legal notes
=================
| SPDX-FileCopyrightText: © 2022 ekvip automation GmbH <info@ekvip.de>
| SPDX-License-Identifier: Apache-2.0
| For details check: Apache-2.0_

.. _Apache-2.0: https://www.apache.org/licenses/LICENSE-2.0

.. _Apache-2.THIS^.SIZE_ZERO: https://www.apache.org/licenses/LICENSE-2.THIS^.SIZE_ZERO

.. </legal notes>

*)

METHOD runIsDwordAlignedTests
VAR
	foo				:XWORD;
	stackAddress	:PVOID;
END_VAR
VAR CONSTANT
	aDWord :DWORD := 16#4;
END_VAR
RETURN (NOT TcUnit.TEST_ORDERED(THIS^.getTestNameFor('isDwordAligned')));
stackAddress := ADR(foo);

THIS^.testIsDwordAligned(
	address := THIS,
);
THIS^.testIsDwordAligned(
	address := THIS^.NULL_POINTER,
);
THIS^.testIsDwordAligned(
	address := THIS^.NULL_POINTER + 1,
);
THIS^.testIsDwordAligned(
	address := stackAddress,
);
THIS^.testIsDwordAligned(
	address := stackAddress + 3,
);
THIS^.testIsDwordAligned(
	address := THIS^.oneByte,
);
THIS^.testIsDwordAligned(
	address := THIS^.oneByte + 7,
);
THIS^.testIsDwordAligned(
	address := THIS^.byteArray,
);
THIS^.testIsDwordAligned(
	address := THIS^.byteArray + 2,
);
THIS^.testIsDwordAligned(
	address := THIS^.cncAddress,
);
THIS^.testIsDwordAligned(
	address := THIS^.cncAddress + 1,
);
THIS^.testIsDwordAligned(
	address := THIS^.itsMeAgain,
);
THIS^.testIsDwordAligned(
	address := THIS^.itsMeAgain + 6,
);
THIS^.testIsDwordAligned(
	address := THIS^.me,
);
THIS^.testIsDwordAligned(
	address := THIS^.me + 3,
);
THIS^.testIsDwordAligned(
	address := THIS^.myMom,
);
THIS^.testIsDwordAligned(
	address := THIS^.invalidByte,
);
THIS^.testIsDwordAligned(
	address := THIS^.invalidByte + 4,
);
THIS^.testIsDwordAligned(
	address := THIS^.INVALID_POINTER,
);
THIS^.testIsDwordAligned(
	address := THIS^.INVALID_POINTER + 1,
);
THIS^.testIsDwordAligned(
	address := aDWord,
);
THIS^.testIsDwordAligned(
	address := aDWord + 1,
);
THIS^.testIsDwordAligned(
	address := TO_DWORD(aDWord - 1),
);

TcUnit.TEST_FINISHED();
END_METHOD

(*

short summary
==================
This test method tests ``assert.pointers.isEqualTo``
method of CNM_AssertionInterfaces library with various inputs

.. <legal notes>

legal notes
=================
| SPDX-FileCopyrightText: © 2022 ekvip automation GmbH <info@ekvip.de>
| SPDX-License-Identifier: Apache-2.0
| For details check: Apache-2.0_

.. _Apache-2.0: https://www.apache.org/licenses/LICENSE-2.0

.. </legal notes>

*)

METHOD runIsEqualToTests
VAR
	foo				:__XWORD;
	stackAddress	:PVOID;
END_VAR
RETURN (NOT TcUnit.TEST_ORDERED(THIS^.getTestNameFor('isEqualTo')));
stackAddress := ADR(foo);
THIS^.testIsEqualTo(
	address1 := THIS,
	address2 := THIS
);
THIS^.testIsEqualTo(
	address1 := THIS^.NULL_POINTER,
	address2 := THIS^.NULL_POINTER
);
THIS^.testIsEqualTo(
	address1 := stackAddress,
	address2 := stackAddress
);
THIS^.testIsEqualTo(
	address1 := THIS^.oneByte,
	address2 := THIS^.oneByte
);
THIS^.testIsEqualTo(
	address1 := THIS^.byteArray,
	address2 := THIS^.byteArray
);
THIS^.testIsEqualTo(
	address1 := THIS^.cncAddress,
	address2 := THIS^.cncAddress
);
THIS^.testIsEqualTo(
	address1 := THIS^.itsMeAgain,
	address2 := THIS^.itsMeAgain
);
THIS^.testIsEqualTo(
	address1 := THIS^.itsMeAgain^,
	address2 := THIS^.itsMeAgain^
);
THIS^.testIsEqualTo(
	address1 := THIS^.me,
	address2 := THIS
);

THIS^.testIsEqualTo(
	address1 := THIS^.itsMeAgain,
	address2 := THIS
);
THIS^.testIsEqualTo(
	address1 := THIS,
	address2 := THIS^.NULL_POINTER
);
THIS^.testIsEqualTo(
	address1 := THIS^.NULL_POINTER,
	address2 := stackAddress
);
THIS^.testIsEqualTo(
	address1 := stackAddress,
	address2 := THIS^.oneByte
);
THIS^.testIsEqualTo(
	address1 := THIS^.oneByte,
	address2 := THIS^.byteArray
);
THIS^.testIsEqualTo(
	address1 := THIS^.byteArray,
	address2 := THIS^.cncAddress
);
THIS^.testIsEqualTo(
	address1 := THIS^.itsMeAgain,
	address2 := THIS^.itsMeAgain
);
THIS^.testIsEqualTo(
	address1 := THIS^.cncAddress,
	address2 := THIS^.itsMeAgain^
);
THIS^.testIsEqualTo(
	address1 := THIS^.itsMeAgain^,
	address2 := THIS^.itsMeAgain
);
THIS^.testIsEqualTo(
	address1 := THIS^.itsMeAgain,
	address2 := THIS
);

TcUnit.TEST_FINISHED();
END_METHOD

(*

short summary
==================
This test method tests ``assert.pointers.isLwordAligned``
method of CNM_AssertionInterfaces library with various inputs

.. <legal notes>

legal notes
=================
| SPDX-FileCopyrightText: © 2022 ekvip automation GmbH <info@ekvip.de>
| SPDX-License-Identifier: Apache-2.0
| For details check: Apache-2.0_

.. _Apache-2.0: https://www.apache.org/licenses/LICENSE-2.0

.. _Apache-2.THIS^.SIZE_ZERO: https://www.apache.org/licenses/LICENSE-2.THIS^.SIZE_ZERO

.. </legal notes>

*)

METHOD runIsLwordAlignedTests
VAR
	foo				:XWORD;
	stackAddress	:PVOID;
	anLword :DWORD := 16#8;
END_VAR
RETURN (NOT TcUnit.TEST_ORDERED(THIS^.getTestNameFor('isLwordAligned')));
stackAddress := ADR(foo);

THIS^.testIsLwordAligned(
	address := THIS,
);
THIS^.testIsLwordAligned(
	address := THIS^.NULL_POINTER,
);
THIS^.testIsLwordAligned(
	address := THIS^.NULL_POINTER + 1,
);
THIS^.testIsLwordAligned(
	address := stackAddress,
);
THIS^.testIsLwordAligned(
	address := stackAddress + 3,
);
THIS^.testIsLwordAligned(
	address := THIS^.oneByte,
);
THIS^.testIsLwordAligned(
	address := THIS^.oneByte + 7,
);
THIS^.testIsLwordAligned(
	address := THIS^.byteArray,
);
THIS^.testIsLwordAligned(
	address := THIS^.byteArray + 2,
);
THIS^.testIsLwordAligned(
	address := THIS^.cncAddress,
);
THIS^.testIsLwordAligned(
	address := THIS^.cncAddress + 1,
);
THIS^.testIsLwordAligned(
	address := THIS^.itsMeAgain,
);
THIS^.testIsLwordAligned(
	address := THIS^.itsMeAgain + 6,
);
THIS^.testIsLwordAligned(
	address := THIS^.me,
);
THIS^.testIsLwordAligned(
	address := THIS^.me + 3,
);
THIS^.testIsLwordAligned(
	address := THIS^.myMom,
);
THIS^.testIsLwordAligned(
	address := THIS^.invalidByte,
);
THIS^.testIsLwordAligned(
	address := THIS^.invalidByte + 4,
);
THIS^.testIsLwordAligned(
	address := THIS^.INVALID_POINTER,
);
THIS^.testIsLwordAligned(
	address := THIS^.INVALID_POINTER + 1,
);
THIS^.testIsLwordAligned(
	address := anLword,
);
THIS^.testIsLwordAligned(
	address := anLword + 1,
);
THIS^.testIsLwordAligned(
	address := anLword - 1,
);

TcUnit.TEST_FINISHED();
END_METHOD

(*

short summary
==================
This test method tests ``assert.pointers.isNotEqualTo``
method of CNM_AssertionInterfaces library with various inputs

.. <legal notes>

legal notes
=================
| SPDX-FileCopyrightText: © 2022 ekvip automation GmbH <info@ekvip.de>
| SPDX-License-Identifier: Apache-2.0
| For details check: Apache-2.0_

.. _Apache-2.0: https://www.apache.org/licenses/LICENSE-2.0

.. </legal notes>

*)

METHOD runIsNotEqualToTests
VAR
	foo				:__XWORD;
	stackAddress	:PVOID;
END_VAR
RETURN (NOT TcUnit.TEST_ORDERED(THIS^.getTestNameFor('isNotEqualTo')));
stackAddress := ADR(foo);
THIS^.testNotIsEqualTo(
	address1 := THIS,
	address2 := THIS
);
THIS^.testNotIsEqualTo(
	address1 := THIS^.NULL_POINTER,
	address2 := THIS^.NULL_POINTER
);
THIS^.testNotIsEqualTo(
	address1 := stackAddress,
	address2 := stackAddress
);
THIS^.testNotIsEqualTo(
	address1 := THIS^.oneByte,
	address2 := THIS^.oneByte
);
THIS^.testNotIsEqualTo(
	address1 := THIS^.byteArray,
	address2 := THIS^.byteArray
);
THIS^.testNotIsEqualTo(
	address1 := THIS^.cncAddress,
	address2 := THIS^.cncAddress
);
THIS^.testNotIsEqualTo(
	address1 := THIS^.itsMeAgain,
	address2 := THIS^.itsMeAgain
);
THIS^.testNotIsEqualTo(
	address1 := THIS^.itsMeAgain^,
	address2 := THIS^.itsMeAgain^
);
THIS^.testNotIsEqualTo(
	address1 := THIS^.me,
	address2 := THIS
);

THIS^.testNotIsEqualTo(
	address1 := THIS^.itsMeAgain,
	address2 := THIS
);
THIS^.testNotIsEqualTo(
	address1 := THIS,
	address2 := THIS^.NULL_POINTER
);
THIS^.testNotIsEqualTo(
	address1 := THIS^.NULL_POINTER,
	address2 := stackAddress
);
THIS^.testNotIsEqualTo(
	address1 := stackAddress,
	address2 := THIS^.oneByte
);
THIS^.testNotIsEqualTo(
	address1 := THIS^.oneByte,
	address2 := THIS^.byteArray
);
THIS^.testNotIsEqualTo(
	address1 := THIS^.byteArray,
	address2 := THIS^.cncAddress
);
THIS^.testNotIsEqualTo(
	address1 := THIS^.itsMeAgain,
	address2 := THIS^.itsMeAgain
);
THIS^.testNotIsEqualTo(
	address1 := THIS^.cncAddress,
	address2 := THIS^.itsMeAgain^
);
THIS^.testNotIsEqualTo(
	address1 := THIS^.itsMeAgain^,
	address2 := THIS^.itsMeAgain
);
THIS^.testNotIsEqualTo(
	address1 := THIS^.itsMeAgain,
	address2 := THIS
);

TcUnit.TEST_FINISHED();
END_METHOD

(*

short summary
==================
This test method tests ``assert.pointers.isNotNull``
method of CNM_AssertionInterfaces library with various inputs

.. <legal notes>

legal notes
=================
| SPDX-FileCopyrightText: © 2022 ekvip automation GmbH <info@ekvip.de>
| SPDX-License-Identifier: Apache-2.0
| For details check: Apache-2.0_

.. _Apache-2.0: https://www.apache.org/licenses/LICENSE-2.0

.. </legal notes>

*)

METHOD runIsNotNullTests
VAR
	foo				:__XWORD;
	stackAddress	:PVOID;
END_VAR
RETURN (NOT TcUnit.TEST_ORDERED(THIS^.getTestNameFor('isNotNull')));

stackAddress := ADR(foo);

THIS^.testIsNotNull(
	address := THIS,
	symbol := 'THIS'
);
THIS^.testIsNotNull(
	address := THIS^.NULL_POINTER,
	symbol := 'THIS^.NULL_POINTER'
);
THIS^.testIsNotNull(
	address := stackAddress,
	symbol := 'stackAddress'
);
THIS^.testIsNotNull(
	address := THIS^.oneByte,
	symbol := 'THIS^.oneByte'
);
THIS^.testIsNotNull(
	address := THIS^.byteArray,
	symbol := 'THIS^.byteArray'
);
THIS^.testIsNotNull(
	address := THIS^.cncAddress,
	symbol := 'THIS^.cncAddress'
);
THIS^.testIsNotNull(
	address := THIS^.itsMeAgain,
	symbol := 'THIS^.itsMeAgain'
);
THIS^.testIsNotNull(
	address := THIS^.itsMeAgain^,
	symbol := 'THIS^.itsMeAgain^'
);
THIS^.testIsNotNull(
	address := THIS^.me,
	symbol := 'THIS^.me'
);

TcUnit.TEST_FINISHED();
END_METHOD

(*

short summary
==================
This test method tests ``assert.pointers.isNotOverlapping``
method of CNM_AssertionInterfaces library with various inputs

.. <legal notes>

legal notes
=================
| SPDX-FileCopyrightText: © 2022 ekvip automation GmbH <info@ekvip.de>
| SPDX-License-Identifier: Apache-2.0
| For details check: Apache-2.0_

.. _Apache-2.0: https://www.apache.org/licenses/LICENSE-2.0

.. _Apache-2.THIS^.SIZE_ZERO: https://www.apache.org/licenses/LICENSE-2.THIS^.SIZE_ZERO

.. </legal notes>

*)

METHOD runIsNotOverlappingTests
VAR
	foo				:XWORD;
	stackAddress	:PVOID;
END_VAR
RETURN (NOT TcUnit.TEST_ORDERED(THIS^.getTestNameFor('isNotOverlapping')));
stackAddress := ADR(foo);

THIS^.testisNotOverlapping(
	address1 := THIS,
	sizeInBytes1 := THIS^.I_AM_FAT,
	address2 := THIS,
	sizeInBytes2 := THIS^.I_AM_FAT
);
THIS^.testisNotOverlapping(
	address1 := THIS,
	sizeInBytes1 := THIS^.I_AM_FAT,
	address2 := THIS^.NULL_POINTER,
	sizeInBytes2 := THIS^.SIZE_ZERO
);
THIS^.testisNotOverlapping(
	address1 := THIS^.NULL_POINTER,
	sizeInBytes1 := THIS^.SIZE_ZERO,
	address2 := THIS^.NULL_POINTER,
	sizeInBytes2 := THIS^.SIZE_ZERO
);
THIS^.testisNotOverlapping(
	address1 := THIS^.NULL_POINTER,
	sizeInBytes1 := THIS^.SIZE_ZERO + 1,
	address2 := THIS^.NULL_POINTER + 1,
	sizeInBytes2 := THIS^.SIZE_ZERO
);
THIS^.testisNotOverlapping(
	address1 := stackAddress,
	sizeInBytes1 := THIS^.SIZE_ZERO,
	address2 := THIS^.oneByte,
	sizeInBytes2 := SIZEOF(BYTE)
);
THIS^.testisNotOverlapping(
	address1 := stackAddress,
	sizeInBytes1 := THIS^.SIZE_ZERO,
	address2 := stackAddress + 1,
	sizeInBytes2 := THIS^.SIZE_ZERO
);
THIS^.testisNotOverlapping(
	address1 := THIS^.byteArray,
	sizeInBytes1 := THIS^.ARRAY_SIZE,
	address2 := THIS^.byteArray + SIZEOF(BYTE),
	sizeInBytes2 := THIS^.SIZE_ZERO
);
THIS^.testisNotOverlapping(
	address2 := THIS^.byteArray,
	sizeInBytes2 := THIS^.ARRAY_SIZE,
	address1 := THIS^.byteArray,
	sizeInBytes1 := THIS^.ARRAY_SIZE + SIZEOF(BYTE)
);
THIS^.testisNotOverlapping(
	address1 := THIS^.cncAddress,
	sizeInBytes1 := THIS^.cncSize,
	address2 := THIS^.cncAddress,
	sizeInBytes2 := THIS^.cncSize,
);
THIS^.testisNotOverlapping(
	address1 := THIS^.cncAddress,
	sizeInBytes1 := THIS^.cncSize - 2,
	address2 := THIS^.cncAddress + 2,
	sizeInBytes2 := THIS^.cncSize + 2,
);
THIS^.testisNotOverlapping(
	address1 := THIS^.itsMeAgain,
	sizeInBytes1 := THIS^.I_AM_FAT,
	address2 := THIS,
	sizeInBytes2 := THIS^.I_AM_FAT
);
THIS^.testisNotOverlapping(
	address1 := THIS^.itsMeAgain,
	sizeInBytes1 := THIS^.I_AM_FAT,
	address2 := THIS^.me,
	sizeInBytes2 := THIS^.I_AM_FAT
);
THIS^.testisNotOverlapping(
	address1 := THIS^.itsMeAgain + 2 * SIZEOF(BYTE),
	sizeInBytes1 := THIS^.I_AM_FAT,
	address2 := THIS^.me,
	sizeInBytes2 := THIS^.I_AM_FAT
);
THIS^.testisNotOverlapping(
	address1 := THIS^.myMom,
	sizeInBytes1 := SIZEOF(AbstractAssertorTest),
	address2 := THIS^.me,
	sizeInBytes2 := THIS^.I_AM_FAT
);
THIS^.testisNotOverlapping(
	address1 := THIS^.myMom,
	sizeInBytes1 := SIZEOF(AbstractAssertorTest),
	address2 := THIS^.me,
	sizeInBytes2 := SIZEOF(AbstractAssertorTest) - THIS^.I_AM_FAT
);
THIS^.testisNotOverlapping(
	address1 := THIS^.invalidByte,
	sizeInBytes1 := SIZEOF(BYTE),
	address2 := THIS^.invalidByte,
	sizeInBytes2 := SIZEOF(BYTE)
);
THIS^.testisNotOverlapping(
	address1 := THIS^.invalidByte,
	sizeInBytes1 := SIZEOF(BYTE),
	address2 := THIS^.invalidByte + (2 * SIZEOF(BYTE)),
	sizeInBytes2 := SIZEOF(BYTE)
);
THIS^.testisNotOverlapping(
	address1 := THIS^.INVALID_POINTER,
	sizeInBytes1 := SIZEOF(BYTE),
	address2 := THIS^.INVALID_POINTER,
	sizeInBytes2 := SIZEOF(BYTE)
);

TcUnit.TEST_FINISHED();
END_METHOD

(*

short summary
==================
This test method tests ``assert.pointers.isNull``
method of CNM_AssertionInterfaces library with various inputs

.. <legal notes>

legal notes
=================
| SPDX-FileCopyrightText: © 2022 ekvip automation GmbH <info@ekvip.de>
| SPDX-License-Identifier: Apache-2.0
| For details check: Apache-2.0_

.. _Apache-2.0: https://www.apache.org/licenses/LICENSE-2.0

.. </legal notes>

*)

METHOD runIsNullTests
VAR
	foo				:__XWORD;
	stackAddress	:PVOID;
END_VAR
RETURN (NOT TcUnit.TEST_ORDERED(THIS^.getTestNameFor('isNull')));

stackAddress := ADR(foo);

THIS^.testIsNull(
	address := THIS,
	symbol := 'THIS'
);
THIS^.testIsNull(
	address := THIS^.NULL_POINTER,
	symbol := 'THIS^.NULL_POINTER'
);
THIS^.testIsNull(
	address := stackAddress,
	symbol := 'stackAddress'
);
THIS^.testIsNull(
	address := THIS^.oneByte,
	symbol := 'THIS^.oneByte'
);
THIS^.testIsNull(
	address := THIS^.byteArray,
	symbol := 'THIS^.byteArray'
);
THIS^.testIsNull(
	address := THIS^.cncAddress,
	symbol := 'THIS^.cncAddress'
);
THIS^.testIsNull(
	address := THIS^.itsMeAgain,
	symbol := 'THIS^.itsMeAgain'
);
THIS^.testIsNull(
	address := THIS^.itsMeAgain^,
	symbol := 'THIS^.itsMeAgain^'
);
THIS^.testIsNull(
	address := THIS^.me,
	symbol := 'THIS^.me'
);

TcUnit.TEST_FINISHED();
END_METHOD

(*

short summary
==================
This test method tests ``assert.pointers.isOverlapping``
method of CNM_AssertionInterfaces library with various inputs

.. <legal notes>

legal notes
=================
| SPDX-FileCopyrightText: © 2022 ekvip automation GmbH <info@ekvip.de>
| SPDX-License-Identifier: Apache-2.0
| For details check: Apache-2.0_

.. _Apache-2.0: https://www.apache.org/licenses/LICENSE-2.0

.. _Apache-2.THIS^.SIZE_ZERO: https://www.apache.org/licenses/LICENSE-2.THIS^.SIZE_ZERO

.. </legal notes>

*)

METHOD runIsOverlappingTests
VAR
	foo				:XWORD;
	stackAddress	:PVOID;
END_VAR
RETURN (NOT TcUnit.TEST_ORDERED(THIS^.getTestNameFor('isOverlapping')));
stackAddress := ADR(foo);

THIS^.testIsOverlapping(
	address1 := THIS,
	sizeInBytes1 := THIS^.I_AM_FAT,
	address2 := THIS,
	sizeInBytes2 := THIS^.I_AM_FAT
);
THIS^.testIsOverlapping(
	address1 := THIS,
	sizeInBytes1 := THIS^.I_AM_FAT,
	address2 := THIS^.NULL_POINTER,
	sizeInBytes2 := THIS^.SIZE_ZERO
);
THIS^.testIsOverlapping(
	address1 := THIS^.NULL_POINTER,
	sizeInBytes1 := THIS^.SIZE_ZERO,
	address2 := THIS^.NULL_POINTER,
	sizeInBytes2 := THIS^.SIZE_ZERO
);
THIS^.testIsOverlapping(
	address1 := THIS^.NULL_POINTER,
	sizeInBytes1 := THIS^.SIZE_ZERO + 1,
	address2 := THIS^.NULL_POINTER + 1,
	sizeInBytes2 := THIS^.SIZE_ZERO
);
THIS^.testIsOverlapping(
	address1 := stackAddress,
	sizeInBytes1 := THIS^.SIZE_ZERO,
	address2 := THIS^.oneByte,
	sizeInBytes2 := SIZEOF(BYTE)
);
THIS^.testIsOverlapping(
	address1 := stackAddress,
	sizeInBytes1 := THIS^.SIZE_ZERO,
	address2 := stackAddress + 1,
	sizeInBytes2 := THIS^.SIZE_ZERO
);
THIS^.testIsOverlapping(
	address1 := THIS^.byteArray,
	sizeInBytes1 := THIS^.ARRAY_SIZE,
	address2 := THIS^.byteArray + SIZEOF(BYTE),
	sizeInBytes2 := THIS^.SIZE_ZERO
);
THIS^.testIsOverlapping(
	address2 := THIS^.byteArray,
	sizeInBytes2 := THIS^.ARRAY_SIZE,
	address1 := THIS^.byteArray,
	sizeInBytes1 := THIS^.ARRAY_SIZE + SIZEOF(BYTE)
);
THIS^.testIsOverlapping(
	address1 := THIS^.cncAddress,
	sizeInBytes1 := THIS^.cncSize,
	address2 := THIS^.cncAddress,
	sizeInBytes2 := THIS^.cncSize,
);
THIS^.testIsOverlapping(
	address1 := THIS^.cncAddress,
	sizeInBytes1 := THIS^.cncSize - 2,
	address2 := THIS^.cncAddress + 2,
	sizeInBytes2 := THIS^.cncSize + 2,
);
THIS^.testIsOverlapping(
	address1 := THIS^.itsMeAgain,
	sizeInBytes1 := THIS^.I_AM_FAT,
	address2 := THIS,
	sizeInBytes2 := THIS^.I_AM_FAT
);
THIS^.testIsOverlapping(
	address1 := THIS^.itsMeAgain,
	sizeInBytes1 := THIS^.I_AM_FAT,
	address2 := THIS^.me,
	sizeInBytes2 := THIS^.I_AM_FAT
);
THIS^.testIsOverlapping(
	address1 := THIS^.itsMeAgain + 2 * SIZEOF(BYTE),
	sizeInBytes1 := THIS^.I_AM_FAT,
	address2 := THIS^.me,
	sizeInBytes2 := THIS^.I_AM_FAT
);
THIS^.testIsOverlapping(
	address1 := THIS^.myMom,
	sizeInBytes1 := SIZEOF(AbstractAssertorTest),
	address2 := THIS^.me,
	sizeInBytes2 := THIS^.I_AM_FAT
);
THIS^.testIsOverlapping(
	address1 := THIS^.myMom,
	sizeInBytes1 := SIZEOF(AbstractAssertorTest),
	address2 := THIS^.me,
	sizeInBytes2 := SIZEOF(AbstractAssertorTest) - THIS^.I_AM_FAT
);
THIS^.testIsOverlapping(
	address1 := THIS^.invalidByte,
	sizeInBytes1 := SIZEOF(BYTE),
	address2 := THIS^.invalidByte,
	sizeInBytes2 := SIZEOF(BYTE)
);
THIS^.testIsOverlapping(
	address1 := THIS^.invalidByte,
	sizeInBytes1 := SIZEOF(BYTE),
	address2 := THIS^.invalidByte + (2 * SIZEOF(BYTE)),
	sizeInBytes2 := SIZEOF(BYTE)
);
THIS^.testIsOverlapping(
	address1 := THIS^.INVALID_POINTER,
	sizeInBytes1 := SIZEOF(BYTE),
	address2 := THIS^.INVALID_POINTER,
	sizeInBytes2 := SIZEOF(BYTE)
);

TcUnit.TEST_FINISHED();
END_METHOD

(*

short summary
==================
This test method tests ``assert.pointers.isValid``
method of CNM_AssertionInterfaces library with various inputs

.. <legal notes>

legal notes
=================
| SPDX-FileCopyrightText: © 2022 ekvip automation GmbH <info@ekvip.de>
| SPDX-License-Identifier: Apache-2.0
| For details check: Apache-2.0_

.. _Apache-2.0: https://www.apache.org/licenses/LICENSE-2.0

.. _Apache-2.THIS^.SIZE_ZERO: https://www.apache.org/licenses/LICENSE-2.THIS^.SIZE_ZERO

.. </legal notes>

*)

METHOD runIsValidTests
VAR
	foo				:XWORD;
	stackAddress	:PVOID;
END_VAR
RETURN (NOT TcUnit.TEST_ORDERED(THIS^.getTestNameFor('isValid')));
stackAddress := ADR(foo);

THIS^.testIsValid(
	address := THIS,
	sizeInBytes := THIS^.I_AM_FAT,
	symbol := 'THIS'
);
THIS^.testIsValid(
	address := THIS^.NULL_POINTER,
	sizeInBytes := THIS^.SIZE_ZERO,
	symbol := 'THIS^.NULL_POINTER'
);
THIS^.testIsValid(
	address := stackAddress,
	sizeInBytes := SIZEOF(XWORD),
	symbol := 'stackAddress'
);
THIS^.testIsValid(
	address := THIS^.oneByte,
	sizeInBytes := SIZEOF(BYTE),
	symbol := 'THIS^.oneByte'
);
THIS^.testIsValid(
	address := THIS^.byteArray,
	sizeInBytes := THIS^.ARRAY_SIZE,
	symbol := 'THIS^.byteArray'
);
THIS^.testIsValid(
	address := THIS^.cncAddress,
	sizeInBytes := THIS^.cncSize,
	symbol := 'THIS^.cncAddress'
);
THIS^.testIsValid(
	address := THIS^.itsMeAgain,
	sizeInBytes := SIZEOF(PVOID),
	symbol := 'THIS^.itsMeAgain'
);
THIS^.testIsValid(
	address := THIS^.itsMeAgain^,
	sizeInBytes := THIS^.I_AM_FAT,
	symbol := 'THIS^.itsMeAgain^'
);
THIS^.testIsValid(
	address := THIS^.me,
	sizeInBytes := THIS^.I_AM_FAT,
	symbol := 'THIS^.me'
);
THIS^.testIsValid(
	address := THIS^.myMom,
	sizeInBytes := SIZEOF(AbstractAssertorTest),
	symbol := 'THIS^.myMom'
);
THIS^.testIsValid(
	address := THIS^.invalidByte,
	sizeInBytes := SIZEOF(BYTE),
	symbol := 'THIS^.invalidByte'
);

THIS^.testIsValid(
	address := THIS^.itsMeAgain,
	sizeInBytes := THIS^.SIZE_ZERO,
	symbol := 'THIS^.itsMeAgain'
);
THIS^.testIsValid(
	address := THIS,
	sizeInBytes := THIS^.SIZE_ZERO,
	symbol := 'THIS'
);
THIS^.testIsValid(
	address := THIS^.NULL_POINTER,
	sizeInBytes := SIZEOF(PVOID),
	symbol := 'THIS^.NULL_POINTER'
);
THIS^.testIsValid(
	address := stackAddress,
	sizeInBytes := THIS^.SIZE_ZERO,
	symbol := 'stackAddress'
);
THIS^.testIsValid(
	address := THIS^.oneByte,
	sizeInBytes := THIS^.SIZE_ZERO,
	symbol := 'THIS^.oneByte'
);
THIS^.testIsValid(
	address := THIS^.byteArray,
	sizeInBytes := THIS^.SIZE_ZERO,
	symbol := 'THIS^.byteArray'
);
THIS^.testIsValid(
	address := THIS^.itsMeAgain,
	sizeInBytes := THIS^.SIZE_ZERO,
	symbol := 'THIS^.itsMeAgain'
);
THIS^.testIsValid(
	address := THIS^.cncAddress,
	sizeInBytes := THIS^.SIZE_ZERO,
	symbol := 'THIS^.cncAddress'
);
THIS^.testIsValid(
	address := THIS^.itsMeAgain^,
	sizeInBytes := THIS^.SIZE_ZERO,
	symbol := 'THIS^.itsMeAgain^'
);
THIS^.testIsValid(
	address := THIS^.INVALID_POINTER,
	sizeInBytes := SIZEOF(PVOID),
	symbol := 'THIS^.INVALID_POINTER'
);
THIS^.testIsValid(
	address := THIS^.myMom,
	sizeInBytes := THIS^.SIZE_ZERO,
	symbol := 'THIS^.myMom'
);
THIS^.testIsValid(
	address := THIS^.invalidByte,
	sizeInBytes := THIS^.SIZE_ZERO,
	symbol := 'THIS^.invalidByte'
);

TcUnit.TEST_FINISHED();
END_METHOD

(*

short summary
==================
This test method tests ``assert.pointers.isWordAligned``
method of CNM_AssertionInterfaces library with various inputs

.. <legal notes>

legal notes
=================
| SPDX-FileCopyrightText: © 2022 ekvip automation GmbH <info@ekvip.de>
| SPDX-License-Identifier: Apache-2.0
| For details check: Apache-2.0_

.. _Apache-2.0: https://www.apache.org/licenses/LICENSE-2.0

.. _Apache-2.THIS^.SIZE_ZERO: https://www.apache.org/licenses/LICENSE-2.THIS^.SIZE_ZERO

.. </legal notes>

*)

METHOD runIsWordAlignedTests
VAR
	foo				:XWORD;
	stackAddress	:PVOID;
END_VAR
VAR CONSTANT
	aWord :WORD := 16#2;
END_VAR
RETURN (NOT TcUnit.TEST_ORDERED(THIS^.getTestNameFor('isWordAligned')));
stackAddress := ADR(foo);

THIS^.testIsWordAligned(
	address := THIS,
);
THIS^.testIsWordAligned(
	address := THIS^.NULL_POINTER,
);
THIS^.testIsWordAligned(
	address := THIS^.NULL_POINTER + 1,
);
THIS^.testIsWordAligned(
	address := stackAddress,
);
THIS^.testIsWordAligned(
	address := stackAddress + 3,
);
THIS^.testIsWordAligned(
	address := THIS^.oneByte,
);
THIS^.testIsWordAligned(
	address := THIS^.oneByte + 7,
);
THIS^.testIsWordAligned(
	address := THIS^.byteArray,
);
THIS^.testIsWordAligned(
	address := THIS^.byteArray + 2,
);
THIS^.testIsWordAligned(
	address := THIS^.cncAddress,
);
THIS^.testIsWordAligned(
	address := THIS^.cncAddress + 1,
);
THIS^.testIsWordAligned(
	address := THIS^.itsMeAgain,
);
THIS^.testIsWordAligned(
	address := THIS^.itsMeAgain + 6,
);
THIS^.testIsWordAligned(
	address := THIS^.me,
);
THIS^.testIsWordAligned(
	address := THIS^.me + 3,
);
THIS^.testIsWordAligned(
	address := THIS^.myMom,
);
THIS^.testIsWordAligned(
	address := THIS^.invalidByte,
);
THIS^.testIsWordAligned(
	address := THIS^.invalidByte + 4,
);
THIS^.testIsWordAligned(
	address := THIS^.INVALID_POINTER,
);
THIS^.testIsWordAligned(
	address := THIS^.INVALID_POINTER + 1,
);
THIS^.testIsWordAligned(
	address := aWord,
);
THIS^.testIsWordAligned(
	address := aWord + 1,
);
THIS^.testIsWordAligned(
	address := TO_WORD(aWord - 1),
);

TcUnit.TEST_FINISHED();
END_METHOD

(*

short summary
==================
This test method tests ``assert.pointers.memoryAreaIsCnc``
method of CNM_AssertionInterfaces library with various inputs

.. <legal notes>

legal notes
=================
| SPDX-FileCopyrightText: © 2022 ekvip automation GmbH <info@ekvip.de>
| SPDX-License-Identifier: Apache-2.0
| For details check: Apache-2.0_

.. _Apache-2.0: https://www.apache.org/licenses/LICENSE-2.0

.. _Apache-2.THIS^.SIZE_ZERO: https://www.apache.org/licenses/LICENSE-2.THIS^.SIZE_ZERO

.. </legal notes>

*)

METHOD runMemoryAreaIsCncTests
VAR
	foo				:__XWORD;
	stackAddress	:PVOID;
END_VAR
RETURN (NOT TcUnit.TEST_ORDERED(THIS^.getTestNameFor('memoryAreaIsCnc')));
stackAddress := ADR(foo);

THIS^.testMemoryAreaIsCnc(
	address := THIS,
	sizeInBytes := THIS^.I_AM_FAT,
	symbol := 'THIS'
);
THIS^.testMemoryAreaIsCnc(
	address := THIS^.NULL_POINTER,
	sizeInBytes := THIS^.SIZE_ZERO,
	symbol := 'THIS^.NULL_POINTER'
);
THIS^.testMemoryAreaIsCnc(
	address := stackAddress,
	sizeInBytes := SIZEOF(__XWORD),
	symbol := 'stackAddress'
);
THIS^.testMemoryAreaIsCnc(
	address := THIS^.oneByte,
	sizeInBytes := SIZEOF(BYTE),
	symbol := 'THIS^.oneByte'
);
THIS^.testMemoryAreaIsCnc(
	address := THIS^.byteArray,
	sizeInBytes := THIS^.ARRAY_SIZE,
	symbol := 'THIS^.byteArray'
);
THIS^.testMemoryAreaIsCnc(
	address := THIS^.cncAddress,
	sizeInBytes := THIS^.cncSize,
	symbol := 'THIS^.cncAddress'
);
THIS^.testMemoryAreaIsCnc(
	address := THIS^.itsMeAgain,
	sizeInBytes := SIZEOF(PVOID),
	symbol := 'THIS^.itsMeAgain'
);
THIS^.testMemoryAreaIsCnc(
	address := THIS^.itsMeAgain^,
	sizeInBytes := THIS^.I_AM_FAT,
	symbol := 'THIS^.itsMeAgain^'
);
THIS^.testMemoryAreaIsCnc(
	address := THIS^.me,
	sizeInBytes := THIS^.I_AM_FAT,
	symbol := 'THIS^.me'
);
THIS^.testMemoryAreaIsCnc(
	address := THIS^.myMom,
	sizeInBytes := SIZEOF(AbstractAssertorTest),
	symbol := 'THIS^.myMom'
);
THIS^.testMemoryAreaIsCnc(
	address := THIS^.invalidByte,
	sizeInBytes := SIZEOF(BYTE),
	symbol := 'THIS^.invalidByte'
);

THIS^.testMemoryAreaIsCnc(
	address := THIS^.itsMeAgain,
	sizeInBytes := THIS^.SIZE_ZERO,
	symbol := 'THIS^.itsMeAgain'
);
THIS^.testMemoryAreaIsCnc(
	address := THIS,
	sizeInBytes := THIS^.SIZE_ZERO,
	symbol := 'THIS'
);
THIS^.testMemoryAreaIsCnc(
	address := THIS^.NULL_POINTER,
	sizeInBytes := SIZEOF(PVOID),
	symbol := 'THIS^.NULL_POINTER'
);
THIS^.testMemoryAreaIsCnc(
	address := stackAddress,
	sizeInBytes := THIS^.SIZE_ZERO,
	symbol := 'stackAddress'
);
THIS^.testMemoryAreaIsCnc(
	address := THIS^.oneByte,
	sizeInBytes := THIS^.SIZE_ZERO,
	symbol := 'THIS^.oneByte'
);
THIS^.testMemoryAreaIsCnc(
	address := THIS^.byteArray,
	sizeInBytes := THIS^.SIZE_ZERO,
	symbol := 'THIS^.byteArray'
);
THIS^.testMemoryAreaIsCnc(
	address := THIS^.itsMeAgain,
	sizeInBytes := THIS^.SIZE_ZERO,
	symbol := 'THIS^.itsMeAgain'
);
THIS^.testMemoryAreaIsCnc(
	address := THIS^.cncAddress,
	sizeInBytes := THIS^.SIZE_ZERO,
	symbol := 'THIS^.cncAddress'
);
THIS^.testMemoryAreaIsCnc(
	address := THIS^.itsMeAgain^,
	sizeInBytes := THIS^.SIZE_ZERO,
	symbol := 'THIS^.itsMeAgain^'
);
THIS^.testMemoryAreaIsCnc(
	address := THIS^.INVALID_POINTER,
	sizeInBytes := SIZEOF(PVOID),
	symbol := 'THIS^.INVALID_POINTER'
);
THIS^.testMemoryAreaIsCnc(
	address := THIS^.myMom,
	sizeInBytes := THIS^.SIZE_ZERO,
	symbol := 'THIS^.myMom'
);
THIS^.testMemoryAreaIsCnc(
	address := THIS^.invalidByte,
	sizeInBytes := THIS^.SIZE_ZERO,
	symbol := 'THIS^.invalidByte'
);

TcUnit.TEST_FINISHED();
END_METHOD

(*

short summary
==================
This test method tests ``assert.pointers.memoryAreaIsDynamic``
method of CNM_AssertionInterfaces library with various inputs

.. <legal notes>

legal notes
=================
| SPDX-FileCopyrightText: © 2022 ekvip automation GmbH <info@ekvip.de>
| SPDX-License-Identifier: Apache-2.0
| For details check: Apache-2.0_

.. _Apache-2.0: https://www.apache.org/licenses/LICENSE-2.0

.. _Apache-2.THIS^.SIZE_ZERO: https://www.apache.org/licenses/LICENSE-2.THIS^.SIZE_ZERO

.. </legal notes>

*)

METHOD runMemoryAreaIsDynamicTests
VAR
	foo				:__XWORD;
	stackAddress	:PVOID;
END_VAR
RETURN (NOT TcUnit.TEST_ORDERED(THIS^.getTestNameFor('memoryAreaIsDynamic')));
stackAddress := ADR(foo);

THIS^.testMemoryAreaIsDynamic(
	address := THIS,
	sizeInBytes := THIS^.I_AM_FAT,
	symbol := 'THIS'
);
THIS^.testMemoryAreaIsDynamic(
	address := THIS^.NULL_POINTER,
	sizeInBytes := THIS^.SIZE_ZERO,
	symbol := 'THIS^.NULL_POINTER'
);
THIS^.testMemoryAreaIsDynamic(
	address := stackAddress,
	sizeInBytes := SIZEOF(__XWORD),
	symbol := 'stackAddress'
);
THIS^.testMemoryAreaIsDynamic(
	address := THIS^.oneByte,
	sizeInBytes := SIZEOF(BYTE),
	symbol := 'THIS^.oneByte'
);
THIS^.testMemoryAreaIsDynamic(
	address := THIS^.byteArray,
	sizeInBytes := THIS^.ARRAY_SIZE,
	symbol := 'THIS^.byteArray'
);
THIS^.testMemoryAreaIsDynamic(
	address := THIS^.cncAddress,
	sizeInBytes := THIS^.cncSize,
	symbol := 'THIS^.cncAddress'
);
THIS^.testMemoryAreaIsDynamic(
	address := THIS^.itsMeAgain,
	sizeInBytes := SIZEOF(PVOID),
	symbol := 'THIS^.itsMeAgain'
);
THIS^.testMemoryAreaIsDynamic(
	address := THIS^.itsMeAgain^,
	sizeInBytes := THIS^.I_AM_FAT,
	symbol := 'THIS^.itsMeAgain^'
);
THIS^.testMemoryAreaIsDynamic(
	address := THIS^.me,
	sizeInBytes := THIS^.I_AM_FAT,
	symbol := 'THIS^.me'
);
THIS^.testMemoryAreaIsDynamic(
	address := THIS^.myMom,
	sizeInBytes := SIZEOF(AbstractAssertorTest),
	symbol := 'THIS^.myMom'
);
THIS^.testMemoryAreaIsDynamic(
	address := THIS^.invalidByte,
	sizeInBytes := SIZEOF(BYTE),
	symbol := 'THIS^.invalidByte'
);

THIS^.testMemoryAreaIsDynamic(
	address := THIS^.itsMeAgain,
	sizeInBytes := THIS^.SIZE_ZERO,
	symbol := 'THIS^.itsMeAgain'
);
THIS^.testMemoryAreaIsDynamic(
	address := THIS,
	sizeInBytes := THIS^.SIZE_ZERO,
	symbol := 'THIS'
);
THIS^.testMemoryAreaIsDynamic(
	address := THIS^.NULL_POINTER,
	sizeInBytes := SIZEOF(PVOID),
	symbol := 'THIS^.NULL_POINTER'
);
THIS^.testMemoryAreaIsDynamic(
	address := stackAddress,
	sizeInBytes := THIS^.SIZE_ZERO,
	symbol := 'stackAddress'
);
THIS^.testMemoryAreaIsDynamic(
	address := THIS^.oneByte,
	sizeInBytes := THIS^.SIZE_ZERO,
	symbol := 'THIS^.oneByte'
);
THIS^.testMemoryAreaIsDynamic(
	address := THIS^.byteArray,
	sizeInBytes := THIS^.SIZE_ZERO,
	symbol := 'THIS^.byteArray'
);
THIS^.testMemoryAreaIsDynamic(
	address := THIS^.itsMeAgain,
	sizeInBytes := THIS^.SIZE_ZERO,
	symbol := 'THIS^.itsMeAgain'
);
THIS^.testMemoryAreaIsDynamic(
	address := THIS^.cncAddress,
	sizeInBytes := THIS^.SIZE_ZERO,
	symbol := 'THIS^.cncAddress'
);
THIS^.testMemoryAreaIsDynamic(
	address := THIS^.itsMeAgain^,
	sizeInBytes := THIS^.SIZE_ZERO,
	symbol := 'THIS^.itsMeAgain^'
);
THIS^.testMemoryAreaIsDynamic(
	address := THIS^.INVALID_POINTER,
	sizeInBytes := SIZEOF(PVOID),
	symbol := 'THIS^.INVALID_POINTER'
);
THIS^.testMemoryAreaIsDynamic(
	address := THIS^.myMom,
	sizeInBytes := THIS^.SIZE_ZERO,
	symbol := 'THIS^.myMom'
);
THIS^.testMemoryAreaIsDynamic(
	address := THIS^.invalidByte,
	sizeInBytes := THIS^.SIZE_ZERO,
	symbol := 'THIS^.invalidByte'
);

TcUnit.TEST_FINISHED();
END_METHOD

(*

short summary
==================
This test method tests ``assert.pointers.memoryAreaIsNotCnc``
method of CNM_AssertionInterfaces library with various inputs

.. <legal notes>

legal notes
=================
| SPDX-FileCopyrightText: © 2022 ekvip automation GmbH <info@ekvip.de>
| SPDX-License-Identifier: Apache-2.0
| For details check: Apache-2.0_

.. _Apache-2.0: https://www.apache.org/licenses/LICENSE-2.0

.. _Apache-2.THIS^.SIZE_ZERO: https://www.apache.org/licenses/LICENSE-2.THIS^.SIZE_ZERO

.. </legal notes>

*)

METHOD runMemoryAreaIsNotCncTests
VAR
	foo				:__XWORD;
	stackAddress	:PVOID;
END_VAR
RETURN (NOT TcUnit.TEST_ORDERED(THIS^.getTestNameFor('memoryAreaIsNotCnc')));
stackAddress := ADR(foo);

THIS^.testMemoryAreaIsNotCnc(
	address := THIS,
	sizeInBytes := THIS^.I_AM_FAT,
	symbol := 'THIS'
);
THIS^.testMemoryAreaIsNotCnc(
	address := THIS^.NULL_POINTER,
	sizeInBytes := THIS^.SIZE_ZERO,
	symbol := 'THIS^.NULL_POINTER'
);
THIS^.testMemoryAreaIsNotCnc(
	address := stackAddress,
	sizeInBytes := SIZEOF(__XWORD),
	symbol := 'stackAddress'
);
THIS^.testMemoryAreaIsNotCnc(
	address := THIS^.oneByte,
	sizeInBytes := SIZEOF(BYTE),
	symbol := 'THIS^.oneByte'
);
THIS^.testMemoryAreaIsNotCnc(
	address := THIS^.byteArray,
	sizeInBytes := THIS^.ARRAY_SIZE,
	symbol := 'THIS^.byteArray'
);
THIS^.testMemoryAreaIsNotCnc(
	address := THIS^.cncAddress,
	sizeInBytes := THIS^.cncSize,
	symbol := 'THIS^.cncAddress'
);
THIS^.testMemoryAreaIsNotCnc(
	address := THIS^.itsMeAgain,
	sizeInBytes := SIZEOF(PVOID),
	symbol := 'THIS^.itsMeAgain'
);
THIS^.testMemoryAreaIsNotCnc(
	address := THIS^.itsMeAgain^,
	sizeInBytes := THIS^.I_AM_FAT,
	symbol := 'THIS^.itsMeAgain^'
);
THIS^.testMemoryAreaIsNotCnc(
	address := THIS^.me,
	sizeInBytes := THIS^.I_AM_FAT,
	symbol := 'THIS^.me'
);
THIS^.testMemoryAreaIsNotCnc(
	address := THIS^.myMom,
	sizeInBytes := SIZEOF(AbstractAssertorTest),
	symbol := 'THIS^.myMom'
);
THIS^.testMemoryAreaIsNotCnc(
	address := THIS^.invalidByte,
	sizeInBytes := SIZEOF(BYTE),
	symbol := 'THIS^.invalidByte'
);

THIS^.testMemoryAreaIsNotCnc(
	address := THIS^.itsMeAgain,
	sizeInBytes := THIS^.SIZE_ZERO,
	symbol := 'THIS^.itsMeAgain'
);
THIS^.testMemoryAreaIsNotCnc(
	address := THIS,
	sizeInBytes := THIS^.SIZE_ZERO,
	symbol := 'THIS'
);
THIS^.testMemoryAreaIsNotCnc(
	address := THIS^.NULL_POINTER,
	sizeInBytes := SIZEOF(PVOID),
	symbol := 'THIS^.NULL_POINTER'
);
THIS^.testMemoryAreaIsNotCnc(
	address := stackAddress,
	sizeInBytes := THIS^.SIZE_ZERO,
	symbol := 'stackAddress'
);
THIS^.testMemoryAreaIsNotCnc(
	address := THIS^.oneByte,
	sizeInBytes := THIS^.SIZE_ZERO,
	symbol := 'THIS^.oneByte'
);
THIS^.testMemoryAreaIsNotCnc(
	address := THIS^.byteArray,
	sizeInBytes := THIS^.SIZE_ZERO,
	symbol := 'THIS^.byteArray'
);
THIS^.testMemoryAreaIsNotCnc(
	address := THIS^.itsMeAgain,
	sizeInBytes := THIS^.SIZE_ZERO,
	symbol := 'THIS^.itsMeAgain'
);
THIS^.testMemoryAreaIsNotCnc(
	address := THIS^.cncAddress,
	sizeInBytes := THIS^.SIZE_ZERO,
	symbol := 'THIS^.cncAddress'
);
THIS^.testMemoryAreaIsNotCnc(
	address := THIS^.itsMeAgain^,
	sizeInBytes := THIS^.SIZE_ZERO,
	symbol := 'THIS^.itsMeAgain^'
);
THIS^.testMemoryAreaIsNotCnc(
	address := THIS^.INVALID_POINTER,
	sizeInBytes := SIZEOF(PVOID),
	symbol := 'THIS^.INVALID_POINTER'
);
THIS^.testMemoryAreaIsNotCnc(
	address := THIS^.myMom,
	sizeInBytes := THIS^.SIZE_ZERO,
	symbol := 'THIS^.myMom'
);
THIS^.testMemoryAreaIsNotCnc(
	address := THIS^.invalidByte,
	sizeInBytes := THIS^.SIZE_ZERO,
	symbol := 'THIS^.invalidByte'
);

TcUnit.TEST_FINISHED();
END_METHOD

(*

short summary
==================
This test method tests ``assert.pointers.memoryAreaIsNotDynamic``
method of CNM_AssertionInterfaces library with various inputs

.. <legal notes>

legal notes
=================
| SPDX-FileCopyrightText: © 2022 ekvip automation GmbH <info@ekvip.de>
| SPDX-License-Identifier: Apache-2.0
| For details check: Apache-2.0_

.. _Apache-2.0: https://www.apache.org/licenses/LICENSE-2.0

.. _Apache-2.THIS^.SIZE_ZERO: https://www.apache.org/licenses/LICENSE-2.THIS^.SIZE_ZERO

.. </legal notes>

*)

METHOD runMemoryAreaIsNotDynamicTests
VAR
	foo				:__XWORD;
	stackAddress	:PVOID;
END_VAR
RETURN (NOT TcUnit.TEST_ORDERED(THIS^.getTestNameFor('memoryAreaIsNotDynamic')));
stackAddress := ADR(foo);

THIS^.testMemoryAreaIsNotDynamic(
	address := THIS,
	sizeInBytes := THIS^.I_AM_FAT,
	symbol := 'THIS'
);
THIS^.testMemoryAreaIsNotDynamic(
	address := THIS^.NULL_POINTER,
	sizeInBytes := THIS^.SIZE_ZERO,
	symbol := 'THIS^.NULL_POINTER'
);
THIS^.testMemoryAreaIsNotDynamic(
	address := stackAddress,
	sizeInBytes := SIZEOF(__XWORD),
	symbol := 'stackAddress'
);
THIS^.testMemoryAreaIsNotDynamic(
	address := THIS^.oneByte,
	sizeInBytes := SIZEOF(BYTE),
	symbol := 'THIS^.oneByte'
);
THIS^.testMemoryAreaIsNotDynamic(
	address := THIS^.byteArray,
	sizeInBytes := THIS^.ARRAY_SIZE,
	symbol := 'THIS^.byteArray'
);
THIS^.testMemoryAreaIsNotDynamic(
	address := THIS^.cncAddress,
	sizeInBytes := THIS^.cncSize,
	symbol := 'THIS^.cncAddress'
);
THIS^.testMemoryAreaIsNotDynamic(
	address := THIS^.itsMeAgain,
	sizeInBytes := SIZEOF(PVOID),
	symbol := 'THIS^.itsMeAgain'
);
THIS^.testMemoryAreaIsNotDynamic(
	address := THIS^.itsMeAgain^,
	sizeInBytes := THIS^.I_AM_FAT,
	symbol := 'THIS^.itsMeAgain^'
);
THIS^.testMemoryAreaIsNotDynamic(
	address := THIS^.me,
	sizeInBytes := THIS^.I_AM_FAT,
	symbol := 'THIS^.me'
);
THIS^.testMemoryAreaIsNotDynamic(
	address := THIS^.myMom,
	sizeInBytes := SIZEOF(AbstractAssertorTest),
	symbol := 'THIS^.myMom'
);
THIS^.testMemoryAreaIsNotDynamic(
	address := THIS^.invalidByte,
	sizeInBytes := SIZEOF(BYTE),
	symbol := 'THIS^.invalidByte'
);

THIS^.testMemoryAreaIsNotDynamic(
	address := THIS^.itsMeAgain,
	sizeInBytes := THIS^.SIZE_ZERO,
	symbol := 'THIS^.itsMeAgain'
);
THIS^.testMemoryAreaIsNotDynamic(
	address := THIS,
	sizeInBytes := THIS^.SIZE_ZERO,
	symbol := 'THIS'
);
THIS^.testMemoryAreaIsNotDynamic(
	address := THIS^.NULL_POINTER,
	sizeInBytes := SIZEOF(PVOID),
	symbol := 'THIS^.NULL_POINTER'
);
THIS^.testMemoryAreaIsNotDynamic(
	address := stackAddress,
	sizeInBytes := THIS^.SIZE_ZERO,
	symbol := 'stackAddress'
);
THIS^.testMemoryAreaIsNotDynamic(
	address := THIS^.oneByte,
	sizeInBytes := THIS^.SIZE_ZERO,
	symbol := 'THIS^.oneByte'
);
THIS^.testMemoryAreaIsNotDynamic(
	address := THIS^.byteArray,
	sizeInBytes := THIS^.SIZE_ZERO,
	symbol := 'THIS^.byteArray'
);
THIS^.testMemoryAreaIsNotDynamic(
	address := THIS^.itsMeAgain,
	sizeInBytes := THIS^.SIZE_ZERO,
	symbol := 'THIS^.itsMeAgain'
);
THIS^.testMemoryAreaIsNotDynamic(
	address := THIS^.cncAddress,
	sizeInBytes := THIS^.SIZE_ZERO,
	symbol := 'THIS^.cncAddress'
);
THIS^.testMemoryAreaIsNotDynamic(
	address := THIS^.itsMeAgain^,
	sizeInBytes := THIS^.SIZE_ZERO,
	symbol := 'THIS^.itsMeAgain^'
);
THIS^.testMemoryAreaIsNotDynamic(
	address := THIS^.INVALID_POINTER,
	sizeInBytes := SIZEOF(PVOID),
	symbol := 'THIS^.INVALID_POINTER'
);
THIS^.testMemoryAreaIsNotDynamic(
	address := THIS^.myMom,
	sizeInBytes := THIS^.SIZE_ZERO,
	symbol := 'THIS^.myMom'
);
THIS^.testMemoryAreaIsNotDynamic(
	address := THIS^.invalidByte,
	sizeInBytes := THIS^.SIZE_ZERO,
	symbol := 'THIS^.invalidByte'
);

TcUnit.TEST_FINISHED();
END_METHOD

(*

short summary
==================
This test method tests ``assert.pointers.memoryAreaIsNotStatic``
method of CNM_AssertionInterfaces library with various inputs

.. <legal notes>

legal notes
=================
| SPDX-FileCopyrightText: © 2022 ekvip automation GmbH <info@ekvip.de>
| SPDX-License-Identifier: Apache-2.0
| For details check: Apache-2.0_

.. _Apache-2.0: https://www.apache.org/licenses/LICENSE-2.0

.. _Apache-2.THIS^.SIZE_ZERO: https://www.apache.org/licenses/LICENSE-2.THIS^.SIZE_ZERO

.. </legal notes>

*)

METHOD runMemoryAreaIsNotStaticTests
VAR
	foo				:__XWORD;
	stackAddress	:PVOID;
END_VAR
RETURN (NOT TcUnit.TEST_ORDERED(THIS^.getTestNameFor('memoryAreaIsNotStatic')));
stackAddress := ADR(foo);

THIS^.testMemoryAreaIsNotStatic(
	address := THIS,
	sizeInBytes := THIS^.I_AM_FAT,
	symbol := 'THIS'
);
THIS^.testMemoryAreaIsNotStatic(
	address := THIS^.NULL_POINTER,
	sizeInBytes := THIS^.SIZE_ZERO,
	symbol := 'THIS^.NULL_POINTER'
);
THIS^.testMemoryAreaIsNotStatic(
	address := stackAddress,
	sizeInBytes := SIZEOF(__XWORD),
	symbol := 'stackAddress'
);
THIS^.testMemoryAreaIsNotStatic(
	address := THIS^.oneByte,
	sizeInBytes := SIZEOF(BYTE),
	symbol := 'THIS^.oneByte'
);
THIS^.testMemoryAreaIsNotStatic(
	address := THIS^.byteArray,
	sizeInBytes := THIS^.ARRAY_SIZE,
	symbol := 'THIS^.byteArray'
);
THIS^.testMemoryAreaIsNotStatic(
	address := THIS^.cncAddress,
	sizeInBytes := THIS^.cncSize,
	symbol := 'THIS^.cncAddress'
);
THIS^.testMemoryAreaIsNotStatic(
	address := THIS^.itsMeAgain,
	sizeInBytes := SIZEOF(PVOID),
	symbol := 'THIS^.itsMeAgain'
);
THIS^.testMemoryAreaIsNotStatic(
	address := THIS^.itsMeAgain^,
	sizeInBytes := THIS^.I_AM_FAT,
	symbol := 'THIS^.itsMeAgain^'
);
THIS^.testMemoryAreaIsNotStatic(
	address := THIS^.me,
	sizeInBytes := THIS^.I_AM_FAT,
	symbol := 'THIS^.me'
);
THIS^.testMemoryAreaIsNotStatic(
	address := THIS^.myMom,
	sizeInBytes := SIZEOF(AbstractAssertorTest),
	symbol := 'THIS^.myMom'
);
THIS^.testMemoryAreaIsNotStatic(
	address := THIS^.invalidByte,
	sizeInBytes := SIZEOF(BYTE),
	symbol := 'THIS^.invalidByte'
);

THIS^.testMemoryAreaIsNotStatic(
	address := THIS^.itsMeAgain,
	sizeInBytes := THIS^.SIZE_ZERO,
	symbol := 'THIS^.itsMeAgain'
);
THIS^.testMemoryAreaIsNotStatic(
	address := THIS,
	sizeInBytes := THIS^.SIZE_ZERO,
	symbol := 'THIS'
);
THIS^.testMemoryAreaIsNotStatic(
	address := THIS^.NULL_POINTER,
	sizeInBytes := SIZEOF(PVOID),
	symbol := 'THIS^.NULL_POINTER'
);
THIS^.testMemoryAreaIsNotStatic(
	address := stackAddress,
	sizeInBytes := THIS^.SIZE_ZERO,
	symbol := 'stackAddress'
);
THIS^.testMemoryAreaIsNotStatic(
	address := THIS^.oneByte,
	sizeInBytes := THIS^.SIZE_ZERO,
	symbol := 'THIS^.oneByte'
);
THIS^.testMemoryAreaIsNotStatic(
	address := THIS^.byteArray,
	sizeInBytes := THIS^.SIZE_ZERO,
	symbol := 'THIS^.byteArray'
);
THIS^.testMemoryAreaIsNotStatic(
	address := THIS^.itsMeAgain,
	sizeInBytes := THIS^.SIZE_ZERO,
	symbol := 'THIS^.itsMeAgain'
);
THIS^.testMemoryAreaIsNotStatic(
	address := THIS^.cncAddress,
	sizeInBytes := THIS^.SIZE_ZERO,
	symbol := 'THIS^.cncAddress'
);
THIS^.testMemoryAreaIsNotStatic(
	address := THIS^.itsMeAgain^,
	sizeInBytes := THIS^.SIZE_ZERO,
	symbol := 'THIS^.itsMeAgain^'
);
THIS^.testMemoryAreaIsNotStatic(
	address := THIS^.INVALID_POINTER,
	sizeInBytes := SIZEOF(PVOID),
	symbol := 'THIS^.INVALID_POINTER'
);
THIS^.testMemoryAreaIsNotStatic(
	address := THIS^.myMom,
	sizeInBytes := THIS^.SIZE_ZERO,
	symbol := 'THIS^.myMom'
);
THIS^.testMemoryAreaIsNotStatic(
	address := THIS^.invalidByte,
	sizeInBytes := THIS^.SIZE_ZERO,
	symbol := 'THIS^.invalidByte'
);

TcUnit.TEST_FINISHED();
END_METHOD

(*

short summary
==================
This test method tests ``assert.pointers.memoryAreaIsNotUnkown``
method of CNM_AssertionInterfaces library with various inputs

.. <legal notes>

legal notes
=================
| SPDX-FileCopyrightText: © 2022 ekvip automation GmbH <info@ekvip.de>
| SPDX-License-Identifier: Apache-2.0
| For details check: Apache-2.0_

.. _Apache-2.0: https://www.apache.org/licenses/LICENSE-2.0

.. _Apache-2.THIS^.SIZE_ZERO: https://www.apache.org/licenses/LICENSE-2.THIS^.SIZE_ZERO

.. </legal notes>

*)

METHOD runMemoryAreaIsNotUnknownTests
VAR
	foo				:__XWORD;
	stackAddress	:PVOID;
END_VAR
RETURN (NOT TcUnit.TEST_ORDERED(THIS^.getTestNameFor('memoryAreaIsNotUnkown')));
stackAddress := ADR(foo);

THIS^.testMemoryAreaIsNotUnknown(
	address := THIS,
	sizeInBytes := THIS^.I_AM_FAT,
	symbol := 'THIS'
);
THIS^.testMemoryAreaIsNotUnknown(
	address := THIS^.NULL_POINTER,
	sizeInBytes := THIS^.SIZE_ZERO,
	symbol := 'THIS^.NULL_POINTER'
);
THIS^.testMemoryAreaIsNotUnknown(
	address := stackAddress,
	sizeInBytes := SIZEOF(__XWORD),
	symbol := 'stackAddress'
);
THIS^.testMemoryAreaIsNotUnknown(
	address := THIS^.oneByte,
	sizeInBytes := SIZEOF(BYTE),
	symbol := 'THIS^.oneByte'
);
THIS^.testMemoryAreaIsNotUnknown(
	address := THIS^.byteArray,
	sizeInBytes := THIS^.ARRAY_SIZE,
	symbol := 'THIS^.byteArray'
);
THIS^.testMemoryAreaIsNotUnknown(
	address := THIS^.cncAddress,
	sizeInBytes := THIS^.cncSize,
	symbol := 'THIS^.cncAddress'
);
THIS^.testMemoryAreaIsNotUnknown(
	address := THIS^.itsMeAgain,
	sizeInBytes := SIZEOF(PVOID),
	symbol := 'THIS^.itsMeAgain'
);
THIS^.testMemoryAreaIsNotUnknown(
	address := THIS^.itsMeAgain^,
	sizeInBytes := THIS^.I_AM_FAT,
	symbol := 'THIS^.itsMeAgain^'
);
THIS^.testMemoryAreaIsNotUnknown(
	address := THIS^.me,
	sizeInBytes := THIS^.I_AM_FAT,
	symbol := 'THIS^.me'
);
THIS^.testMemoryAreaIsNotUnknown(
	address := THIS^.myMom,
	sizeInBytes := SIZEOF(AbstractAssertorTest),
	symbol := 'THIS^.myMom'
);
THIS^.testMemoryAreaIsNotUnknown(
	address := THIS^.invalidByte,
	sizeInBytes := SIZEOF(BYTE),
	symbol := 'THIS^.invalidByte'
);

THIS^.testMemoryAreaIsNotUnknown(
	address := THIS^.itsMeAgain,
	sizeInBytes := THIS^.SIZE_ZERO,
	symbol := 'THIS^.itsMeAgain'
);
THIS^.testMemoryAreaIsNotUnknown(
	address := THIS,
	sizeInBytes := THIS^.SIZE_ZERO,
	symbol := 'THIS'
);
THIS^.testMemoryAreaIsNotUnknown(
	address := THIS^.NULL_POINTER,
	sizeInBytes := SIZEOF(PVOID),
	symbol := 'THIS^.NULL_POINTER'
);
THIS^.testMemoryAreaIsNotUnknown(
	address := stackAddress,
	sizeInBytes := THIS^.SIZE_ZERO,
	symbol := 'stackAddress'
);
THIS^.testMemoryAreaIsNotUnknown(
	address := THIS^.oneByte,
	sizeInBytes := THIS^.SIZE_ZERO,
	symbol := 'THIS^.oneByte'
);
THIS^.testMemoryAreaIsNotUnknown(
	address := THIS^.byteArray,
	sizeInBytes := THIS^.SIZE_ZERO,
	symbol := 'THIS^.byteArray'
);
THIS^.testMemoryAreaIsNotUnknown(
	address := THIS^.itsMeAgain,
	sizeInBytes := THIS^.SIZE_ZERO,
	symbol := 'THIS^.itsMeAgain'
);
THIS^.testMemoryAreaIsNotUnknown(
	address := THIS^.cncAddress,
	sizeInBytes := THIS^.SIZE_ZERO,
	symbol := 'THIS^.cncAddress'
);
THIS^.testMemoryAreaIsNotUnknown(
	address := THIS^.itsMeAgain^,
	sizeInBytes := THIS^.SIZE_ZERO,
	symbol := 'THIS^.itsMeAgain^'
);
THIS^.testMemoryAreaIsNotUnknown(
	address := THIS^.INVALID_POINTER,
	sizeInBytes := SIZEOF(PVOID),
	symbol := 'THIS^.INVALID_POINTER'
);
THIS^.testMemoryAreaIsNotUnknown(
	address := THIS^.myMom,
	sizeInBytes := THIS^.SIZE_ZERO,
	symbol := 'THIS^.myMom'
);
THIS^.testMemoryAreaIsNotUnknown(
	address := THIS^.invalidByte,
	sizeInBytes := THIS^.SIZE_ZERO,
	symbol := 'THIS^.invalidByte'
);

TcUnit.TEST_FINISHED();
END_METHOD

(*

short summary
==================
This test method tests ``assert.pointers.memoryAreaIsStatic``
method of CNM_AssertionInterfaces library with various inputs

.. <legal notes>

legal notes
=================
| SPDX-FileCopyrightText: © 2022 ekvip automation GmbH <info@ekvip.de>
| SPDX-License-Identifier: Apache-2.0
| For details check: Apache-2.0_

.. _Apache-2.0: https://www.apache.org/licenses/LICENSE-2.0

.. _Apache-2.THIS^.SIZE_ZERO: https://www.apache.org/licenses/LICENSE-2.THIS^.SIZE_ZERO

.. </legal notes>

*)

METHOD runMemoryAreaIsStaticTests
VAR
	foo				:__XWORD;
	stackAddress	:PVOID;
END_VAR
RETURN (NOT TcUnit.TEST_ORDERED(THIS^.getTestNameFor('memoryAreaIsStatic')));
stackAddress := ADR(foo);

THIS^.testMemoryAreaIsStatic(
	address := THIS,
	sizeInBytes := THIS^.I_AM_FAT,
	symbol := 'THIS'
);
THIS^.testMemoryAreaIsStatic(
	address := THIS^.NULL_POINTER,
	sizeInBytes := THIS^.SIZE_ZERO,
	symbol := 'THIS^.NULL_POINTER'
);
THIS^.testMemoryAreaIsStatic(
	address := stackAddress,
	sizeInBytes := SIZEOF(__XWORD),
	symbol := 'stackAddress'
);
THIS^.testMemoryAreaIsStatic(
	address := THIS^.oneByte,
	sizeInBytes := SIZEOF(BYTE),
	symbol := 'THIS^.oneByte'
);
THIS^.testMemoryAreaIsStatic(
	address := THIS^.byteArray,
	sizeInBytes := THIS^.ARRAY_SIZE,
	symbol := 'THIS^.byteArray'
);
THIS^.testMemoryAreaIsStatic(
	address := THIS^.cncAddress,
	sizeInBytes := THIS^.cncSize,
	symbol := 'THIS^.cncAddress'
);
THIS^.testMemoryAreaIsStatic(
	address := THIS^.itsMeAgain,
	sizeInBytes := SIZEOF(PVOID),
	symbol := 'THIS^.itsMeAgain'
);
THIS^.testMemoryAreaIsStatic(
	address := THIS^.itsMeAgain^,
	sizeInBytes := THIS^.I_AM_FAT,
	symbol := 'THIS^.itsMeAgain^'
);
THIS^.testMemoryAreaIsStatic(
	address := THIS^.me,
	sizeInBytes := THIS^.I_AM_FAT,
	symbol := 'THIS^.me'
);
THIS^.testMemoryAreaIsStatic(
	address := THIS^.myMom,
	sizeInBytes := SIZEOF(AbstractAssertorTest),
	symbol := 'THIS^.myMom'
);
THIS^.testMemoryAreaIsStatic(
	address := THIS^.invalidByte,
	sizeInBytes := SIZEOF(BYTE),
	symbol := 'THIS^.invalidByte'
);

THIS^.testMemoryAreaIsStatic(
	address := THIS^.itsMeAgain,
	sizeInBytes := THIS^.SIZE_ZERO,
	symbol := 'THIS^.itsMeAgain'
);
THIS^.testMemoryAreaIsStatic(
	address := THIS,
	sizeInBytes := THIS^.SIZE_ZERO,
	symbol := 'THIS'
);
THIS^.testMemoryAreaIsStatic(
	address := THIS^.NULL_POINTER,
	sizeInBytes := SIZEOF(PVOID),
	symbol := 'THIS^.NULL_POINTER'
);
THIS^.testMemoryAreaIsStatic(
	address := stackAddress,
	sizeInBytes := THIS^.SIZE_ZERO,
	symbol := 'stackAddress'
);
THIS^.testMemoryAreaIsStatic(
	address := THIS^.oneByte,
	sizeInBytes := THIS^.SIZE_ZERO,
	symbol := 'THIS^.oneByte'
);
THIS^.testMemoryAreaIsStatic(
	address := THIS^.byteArray,
	sizeInBytes := THIS^.SIZE_ZERO,
	symbol := 'THIS^.byteArray'
);
THIS^.testMemoryAreaIsStatic(
	address := THIS^.itsMeAgain,
	sizeInBytes := THIS^.SIZE_ZERO,
	symbol := 'THIS^.itsMeAgain'
);
THIS^.testMemoryAreaIsStatic(
	address := THIS^.cncAddress,
	sizeInBytes := THIS^.SIZE_ZERO,
	symbol := 'THIS^.cncAddress'
);
THIS^.testMemoryAreaIsStatic(
	address := THIS^.itsMeAgain^,
	sizeInBytes := THIS^.SIZE_ZERO,
	symbol := 'THIS^.itsMeAgain^'
);
THIS^.testMemoryAreaIsStatic(
	address := THIS^.INVALID_POINTER,
	sizeInBytes := SIZEOF(PVOID),
	symbol := 'THIS^.INVALID_POINTER'
);
THIS^.testMemoryAreaIsStatic(
	address := THIS^.myMom,
	sizeInBytes := THIS^.SIZE_ZERO,
	symbol := 'THIS^.myMom'
);
THIS^.testMemoryAreaIsStatic(
	address := THIS^.invalidByte,
	sizeInBytes := THIS^.SIZE_ZERO,
	symbol := 'THIS^.invalidByte'
);

TcUnit.TEST_FINISHED();
END_METHOD

(*

short summary
==================
This test method tests ``assert.pointers.memoryAreaIsUnkown``
method of CNM_AssertionInterfaces library with various inputs

.. <legal notes>

legal notes
=================
| SPDX-FileCopyrightText: © 2022 ekvip automation GmbH <info@ekvip.de>
| SPDX-License-Identifier: Apache-2.0
| For details check: Apache-2.0_

.. _Apache-2.0: https://www.apache.org/licenses/LICENSE-2.0

.. _Apache-2.THIS^.SIZE_ZERO: https://www.apache.org/licenses/LICENSE-2.THIS^.SIZE_ZERO

.. </legal notes>

*)

METHOD runMemoryAreaIsUnknownTests
VAR
	foo				:__XWORD;
	stackAddress	:PVOID;
END_VAR
RETURN (NOT TcUnit.TEST_ORDERED(THIS^.getTestNameFor('memoryAreaIsUnkown')));
stackAddress := ADR(foo);

THIS^.testMemoryAreaIsUnknown(
	address := THIS,
	sizeInBytes := THIS^.I_AM_FAT,
	symbol := 'THIS'
);
THIS^.testMemoryAreaIsUnknown(
	address := THIS^.NULL_POINTER,
	sizeInBytes := THIS^.SIZE_ZERO,
	symbol := 'THIS^.NULL_POINTER'
);
THIS^.testMemoryAreaIsUnknown(
	address := stackAddress,
	sizeInBytes := SIZEOF(__XWORD),
	symbol := 'stackAddress'
);
THIS^.testMemoryAreaIsUnknown(
	address := THIS^.oneByte,
	sizeInBytes := SIZEOF(BYTE),
	symbol := 'THIS^.oneByte'
);
THIS^.testMemoryAreaIsUnknown(
	address := THIS^.byteArray,
	sizeInBytes := THIS^.ARRAY_SIZE,
	symbol := 'THIS^.byteArray'
);
THIS^.testMemoryAreaIsUnknown(
	address := THIS^.cncAddress,
	sizeInBytes := THIS^.cncSize,
	symbol := 'THIS^.cncAddress'
);
THIS^.testMemoryAreaIsUnknown(
	address := THIS^.itsMeAgain,
	sizeInBytes := SIZEOF(PVOID),
	symbol := 'THIS^.itsMeAgain'
);
THIS^.testMemoryAreaIsUnknown(
	address := THIS^.itsMeAgain^,
	sizeInBytes := THIS^.I_AM_FAT,
	symbol := 'THIS^.itsMeAgain^'
);
THIS^.testMemoryAreaIsUnknown(
	address := THIS^.me,
	sizeInBytes := THIS^.I_AM_FAT,
	symbol := 'THIS^.me'
);
THIS^.testMemoryAreaIsUnknown(
	address := THIS^.myMom,
	sizeInBytes := SIZEOF(AbstractAssertorTest),
	symbol := 'THIS^.myMom'
);
THIS^.testMemoryAreaIsUnknown(
	address := THIS^.invalidByte,
	sizeInBytes := SIZEOF(BYTE),
	symbol := 'THIS^.invalidByte'
);

THIS^.testMemoryAreaIsUnknown(
	address := THIS^.itsMeAgain,
	sizeInBytes := THIS^.SIZE_ZERO,
	symbol := 'THIS^.itsMeAgain'
);
THIS^.testMemoryAreaIsUnknown(
	address := THIS,
	sizeInBytes := THIS^.SIZE_ZERO,
	symbol := 'THIS'
);
THIS^.testMemoryAreaIsUnknown(
	address := THIS^.NULL_POINTER,
	sizeInBytes := SIZEOF(PVOID),
	symbol := 'THIS^.NULL_POINTER'
);
THIS^.testMemoryAreaIsUnknown(
	address := stackAddress,
	sizeInBytes := THIS^.SIZE_ZERO,
	symbol := 'stackAddress'
);
THIS^.testMemoryAreaIsUnknown(
	address := THIS^.oneByte,
	sizeInBytes := THIS^.SIZE_ZERO,
	symbol := 'THIS^.oneByte'
);
THIS^.testMemoryAreaIsUnknown(
	address := THIS^.byteArray,
	sizeInBytes := THIS^.SIZE_ZERO,
	symbol := 'THIS^.byteArray'
);
THIS^.testMemoryAreaIsUnknown(
	address := THIS^.itsMeAgain,
	sizeInBytes := THIS^.SIZE_ZERO,
	symbol := 'THIS^.itsMeAgain'
);
THIS^.testMemoryAreaIsUnknown(
	address := THIS^.cncAddress,
	sizeInBytes := THIS^.SIZE_ZERO,
	symbol := 'THIS^.cncAddress'
);
THIS^.testMemoryAreaIsUnknown(
	address := THIS^.itsMeAgain^,
	sizeInBytes := THIS^.SIZE_ZERO,
	symbol := 'THIS^.itsMeAgain^'
);
THIS^.testMemoryAreaIsUnknown(
	address := THIS^.INVALID_POINTER,
	sizeInBytes := SIZEOF(PVOID),
	symbol := 'THIS^.INVALID_POINTER'
);
THIS^.testMemoryAreaIsUnknown(
	address := THIS^.myMom,
	sizeInBytes := THIS^.SIZE_ZERO,
	symbol := 'THIS^.myMom'
);
THIS^.testMemoryAreaIsUnknown(
	address := THIS^.invalidByte,
	sizeInBytes := THIS^.SIZE_ZERO,
	symbol := 'THIS^.invalidByte'
);

TcUnit.TEST_FINISHED();
END_METHOD

(*

short summary
==================
This test method tests ``assert.pointers.isAligned``
method of CNM_AssertionInterfaces library, 
it provides the possibility to handover test data via parameter
This test method uses a bit mask to verify correct memory alignment without duplicating the tested function.
(ex. for 64 bit: if bits 0-7 are set, the pointer is not aligned)

.. <legal notes>

legal notes
=================
| SPDX-FileCopyrightText: © 2022 ekvip automation GmbH <info@ekvip.de>
| SPDX-License-Identifier: Apache-2.0
| For details check: Apache-2.0_

.. _Apache-2.0: https://www.apache.org/licenses/LICENSE-2.0

.. </legal notes>

parameters
==========

*)

METHOD testIsAligned
VAR_INPUT
	(* for the test it's the parameter ``address`` *)
	address		:PVOID;
END_VAR
VAR
	(* just the expectation if the assertion to test must be worng or true *)
	assertionIsWrong		:BOOL;
	(* contains the format string for the test message *)
	message					:Tc2_System.T_MaxString;
	(* TwinCAT printf with the test message *)
	messageStringBuilder	:Tc2_Utilities.FB_FormatString;
	(* contains adress of the stack of this method *)
	{attribute 'displaymode':='hex'}
	stackAddress			:__XWORD := ADR(stackAddress);
	(* used to check if pointer is aligned *)
	{attribute 'displaymode':='hex'}
	alignmentMask 			:__UXINT;
END_VAR
THIS^.assertorContainer.resetAssertor();

alignmentMask := XSIZEOF(__XWORD) - 1;

assertionIsWrong := (alignmentMask AND address) <> 0;

message := SEL(
	assertionIsWrong,
	'address is 16#%X and should be aligned, assertion must be TRUE', 
	'address is 16#%X and should not be aligned, assertion must be FALSE'
);
messageStringBuilder(
	sFormat := message,
	arg1 := THIS^.AnyToArg(address),
);

THIS^.assertorContainer.assertor.assert.pointers.isAligned(
	address := address,
	message := ''
);

THIS^.AssertEquals_BOOL(
	Expected 	:= assertionIsWrong,
	Actual 		:= THIS^.assertorContainer.wasAssertionWrong,
	Message 	:= messageStringBuilder.sOut
);
END_METHOD

(*

short summary
==================
This test method tests ``assert.pointers.isDwordAligned``
method of CNM_AssertionInterfaces library, 
it provides the possibility to handover test data via parameter
This test method uses a bit mask to verify correct memory alignment without duplicating the tested function.
(ex. for DWORD: if bits 0-3 are set, the pointer is not aligned)

.. <legal notes>

legal notes
=================
| SPDX-FileCopyrightText: © 2022 ekvip automation GmbH <info@ekvip.de>
| SPDX-License-Identifier: Apache-2.0
| For details check: Apache-2.0_

.. _Apache-2.0: https://www.apache.org/licenses/LICENSE-2.0

.. </legal notes>

parameters
==========

*)

METHOD testIsDwordAligned
VAR_INPUT
	(* for the test it's the parameter ``address`` *)
	address		:PVOID;
END_VAR
VAR
	(* just the expectation if the assertion to test must be worng or true *)
	assertionIsWrong		:BOOL;
	(* contains the format string for the test message *)
	message					:Tc2_System.T_MaxString;
	(* TwinCAT printf with the test message *)
	messageStringBuilder	:Tc2_Utilities.FB_FormatString;
	(* contains adress of the stack of this method *)
	{attribute 'displaymode':='hex'}
	stackAddress			:__XWORD := ADR(stackAddress);
END_VAR
VAR CONSTANT
	(* used to check if pointer is aligned *)
	{attribute 'displaymode':='hex'}
	alignmentMask 			:DWORD := 16#3;
END_VAR
THIS^.assertorContainer.resetAssertor();

assertionIsWrong := (alignmentMask AND address) <> 0;

message := SEL(
	assertionIsWrong,
	'address is 16#%X and should be aligned, assertion must be TRUE', 
	'address is 16#%X and should not be aligned, assertion must be FALSE'
);
messageStringBuilder(
	sFormat := message,
	arg1 := THIS^.AnyToArg(address),
);

THIS^.assertorContainer.assertor.assert.pointers.isDwordAligned(
	address := address,
	message := ''
);

THIS^.AssertEquals_BOOL(
	Expected 	:= assertionIsWrong,
	Actual 		:= THIS^.assertorContainer.wasAssertionWrong,
	Message 	:= messageStringBuilder.sOut
);
END_METHOD

(*

short summary
==================
This test method tests ``assert.pointers.isEqualTo``
method of CNM_AssertionInterfaces library, 
it provides the possibility to handover test data via parameter 


.. <legal notes>

legal notes
=================
| SPDX-FileCopyrightText: © 2022 ekvip automation GmbH <info@ekvip.de>
| SPDX-License-Identifier: Apache-2.0
| For details check: Apache-2.0_

.. _Apache-2.0: https://www.apache.org/licenses/LICENSE-2.0

.. </legal notes>

parameters
==========

*)

METHOD testIsEqualTo
VAR_INPUT
	(* for the test it's the parameter ``address1`` *)
	address1	:PVOID;
	(* for the test it's the parameter ``address2`` *)
	address2	:PVOID;
END_VAR
VAR
	(* just the expectation if the assertion to test must be worng or true *)
	assertionIsWrong		:BOOL;
	(* contains the format string for the test message *)
	message					:Tc2_System.T_MaxString;
	(* TwinCAT printf with the test message *)
	messageStringBuilder	:Tc2_Utilities.FB_FormatString;
END_VAR
THIS^.assertorContainer.resetAssertor();

assertionIsWrong := (address1 <> address2);
message := SEL(
	assertionIsWrong,
	'address1 is 16#%X address2 is 16#%X assertion must be TRUE', 
	'address1 is 16#%X address2 is 16#%X assertion must be FALSE'
);
messageStringBuilder(
	sFormat := message,
	arg1 := THIS^.AnyToArg(address1),
	arg2 := THIS^.AnyToArg(address2)
);

THIS^.assertorContainer.assertor.assert.pointers.isEqualTo(
	address1 := address1,
	address2 := address2,
	message := ''
);

THIS^.AssertEquals_BOOL(
	Expected 	:= assertionIsWrong,
	Actual 		:= THIS^.assertorContainer.wasAssertionWrong,
	Message 	:= messageStringBuilder.sOut
);
END_METHOD

(*

short summary
==================
This test method tests ``assert.pointers.isLwordAligned``
method of CNM_AssertionInterfaces library, 
it provides the possibility to handover test data via parameter
This test method uses a bit mask to verify correct memory alignment without duplicating the tested function.
(ex. for LWORD: if bits 0-7 are set, the pointer is not aligned)

.. <legal notes>

legal notes
=================
| SPDX-FileCopyrightText: © 2022 ekvip automation GmbH <info@ekvip.de>
| SPDX-License-Identifier: Apache-2.0
| For details check: Apache-2.0_

.. _Apache-2.0: https://www.apache.org/licenses/LICENSE-2.0

.. </legal notes>

parameters
==========

*)

METHOD testIsLwordAligned
VAR_INPUT
	(* for the test it's the parameter ``address`` *)
	address		:PVOID;
END_VAR
VAR
	(* just the expectation if the assertion to test must be worng or true *)
	assertionIsWrong		:BOOL;
	(* contains the format string for the test message *)
	message					:Tc2_System.T_MaxString;
	(* TwinCAT printf with the test message *)
	messageStringBuilder	:Tc2_Utilities.FB_FormatString;
	(* contains adress of the stack of this method *)
	{attribute 'displaymode':='hex'}
	stackAddress			:__XWORD := ADR(stackAddress);
END_VAR
VAR CONSTANT
	(* used to check if pointer is aligned *)
	{attribute 'displaymode':='hex'}
	alignmentMask 			:LWORD := 16#7;
END_VAR
THIS^.assertorContainer.resetAssertor();

assertionIsWrong := (alignmentMask AND address) <> 0;

message := SEL(
	assertionIsWrong,
	'address is 16#%X and should be aligned, assertion must be TRUE', 
	'address is 16#%X and should not be aligned, assertion must be FALSE'
);
messageStringBuilder(
	sFormat := message,
	arg1 := THIS^.AnyToArg(address),
);

THIS^.assertorContainer.assertor.assert.pointers.isLwordAligned(
	address := address,
	message := ''
);

THIS^.AssertEquals_BOOL(
	Expected 	:= assertionIsWrong,
	Actual 		:= THIS^.assertorContainer.wasAssertionWrong,
	Message 	:= messageStringBuilder.sOut
);
END_METHOD

(*

short summary
==================
This test method tests ``assert.pointers.isNotNull``
method of CNM_AssertionInterfaces library, 
it provides the possibility to handover test data via parameter 


.. <legal notes>

legal notes
=================
| SPDX-FileCopyrightText: © 2022 ekvip automation GmbH <info@ekvip.de>
| SPDX-License-Identifier: Apache-2.0
| For details check: Apache-2.0_

.. _Apache-2.0: https://www.apache.org/licenses/LICENSE-2.0

.. </legal notes>

parameters
==========

*)

METHOD testIsNotNull
VAR_INPUT
	(* for the test it's the parameter ``address`` *)
	address		:PVOID;
	(* just the name of the pointer *)
	symbol		:Tc2_System.T_MaxString;
END_VAR
VAR
	(* just the expectation if the assertion to test must be worng or true *)
	assertionIsWrong		:BOOL;
	(* contains the format string for the test message *)
	message					:Tc2_System.T_MaxString;
	(* TwinCAT printf with the test message *)
	messageStringBuilder	:Tc2_Utilities.FB_FormatString;
END_VAR
THIS^.assertorContainer.resetAssertor();

assertionIsWrong := (address = THIS^.NULL_POINTER);
message := SEL(
	assertionIsWrong,
	'address is 16#%X ($'%s$') assertion must be TRUE', 
	'address is 16#%X ($'%s$') assertion must be FALSE'
);
messageStringBuilder(
	sFormat := message,
	arg1 := THIS^.AnyToArg(address),
	arg2 := THIS^.AnyToArg(symbol)
);

THIS^.assertorContainer.assertor.assert.pointers.isNotNull(
	address := address,
	message := ''
);

THIS^.AssertEquals_BOOL(
	Expected 	:= assertionIsWrong,
	Actual 		:= THIS^.assertorContainer.wasAssertionWrong,
	Message 	:= messageStringBuilder.sOut
);
END_METHOD

(*

short summary
==================
This test method tests ``assert.pointers.isNotOverlapping``
method of CNM_AssertionInterfaces library, 
it provides the possibility to handover test data via parameter

.. <legal notes>

legal notes
=================
| SPDX-FileCopyrightText: © 2022 ekvip automation GmbH <info@ekvip.de>
| SPDX-License-Identifier: Apache-2.0
| For details check: Apache-2.0_

.. _Apache-2.0: https://www.apache.org/licenses/LICENSE-2.0

.. </legal notes>

parameters
==========

*)

METHOD testIsNotOverlapping
VAR_INPUT
	(* for the test it's the parameter ``address1`` *)
	address1		:PVOID;
	(* for the test it's the parameter ``address2`` *)
	address2		:PVOID;
	(* for the test it's the parameter ``sizeInBytes1`` *)
	sizeInBytes1	:UDINT;
	(* for the test it's the parameter ``sizeInBytes2`` *)
	sizeInBytes2	:UDINT;
END_VAR
VAR
	(* just the expectation if the assertion to test must be worng or true *)
	assertionIsWrong		:BOOL;
	(* contains the format string for the test message *)
	message					:Tc2_System.T_MaxString;
	(* TwinCAT printf with the test message *)
	messageStringBuilder	:Tc2_Utilities.FB_FormatString;
	(* contains adress of the stack of this method *)
	{attribute 'displaymode':='hex'}
	stackAddress			:__XWORD := ADR(stackAddress);
END_VAR
THIS^.assertorContainer.resetAssertor();

assertionIsWrong := address1 + sizeInBytes1 >= address2 
					AND address2 + sizeInBytes2 >= address1;

message := SEL(
	assertionIsWrong,
	'address1 is 16#%X, sizeInBytes is %d and address2 is 16#%X, sizeInBytes is %d, they are not overlapping, assertion must be TRUE', 
	'address1 is 16#%X, sizeInBytes is %d and address2 is 16#%X, sizeInBytes is %d, they are overlapping, assertion must be FALSE'
);
messageStringBuilder(
	sFormat := message,
	arg1 := THIS^.AnyToArg(address1),
	arg1 := THIS^.AnyToArg(sizeInBytes1),
	arg1 := THIS^.AnyToArg(address2),
	arg1 := THIS^.AnyToArg(sizeInBytes2),
);

THIS^.assertorContainer.assertor.assert.pointers.isNotOverlapping(
	address1 := address1,
	address2 := address2,
	sizeInBytes1 := sizeInBytes1,
	sizeInBytes2 := sizeInBytes2,
	message := ''
);

THIS^.AssertEquals_BOOL(
	Expected 	:= assertionIsWrong,
	Actual 		:= THIS^.assertorContainer.wasAssertionWrong,
	Message 	:= messageStringBuilder.sOut
);
END_METHOD

(*

short summary
==================
This test method tests ``assert.pointers.isNull``
method of CNM_AssertionInterfaces library, 
it provides the possibility to handover test data via parameter 


.. <legal notes>

legal notes
=================
| SPDX-FileCopyrightText: © 2022 ekvip automation GmbH <info@ekvip.de>
| SPDX-License-Identifier: Apache-2.0
| For details check: Apache-2.0_

.. _Apache-2.0: https://www.apache.org/licenses/LICENSE-2.0

.. </legal notes>

parameters
==========

*)

METHOD testIsNull
VAR_INPUT
	(* for the test it's the parameter ``address`` *)
	address		:PVOID;
	(* just the name of the pointer *)
	symbol		:Tc2_System.T_MaxString;
END_VAR
VAR
	(* just the expectation if the assertion to test must be worng or true *)
	assertionIsWrong		:BOOL;
	(* contains the format string for the test message *)
	message					:Tc2_System.T_MaxString;
	(* TwinCAT printf with the test message *)
	messageStringBuilder	:Tc2_Utilities.FB_FormatString;
END_VAR
THIS^.assertorContainer.resetAssertor();

assertionIsWrong := (address <> THIS^.NULL_POINTER);
message := SEL(
	assertionIsWrong,
	'address is 16#%X ($'%s$') assertion must be TRUE', 
	'address is 16#%X ($'%s$') assertion must be FALSE'
);
messageStringBuilder(
	sFormat := message,
	arg1 := THIS^.AnyToArg(address),
	arg2 := THIS^.AnyToArg(symbol)
);

THIS^.assertorContainer.assertor.assert.pointers.isNull(
	address := address,
	message := ''
);

THIS^.AssertEquals_BOOL(
	Expected 	:= assertionIsWrong,
	Actual 		:= THIS^.assertorContainer.wasAssertionWrong,
	Message 	:= messageStringBuilder.sOut
);
END_METHOD

(*

short summary
==================
This test method tests ``assert.pointers.isOverlapping``
method of CNM_AssertionInterfaces library, 
it provides the possibility to handover test data via parameter

.. <legal notes>

legal notes
=================
| SPDX-FileCopyrightText: © 2022 ekvip automation GmbH <info@ekvip.de>
| SPDX-License-Identifier: Apache-2.0
| For details check: Apache-2.0_

.. _Apache-2.0: https://www.apache.org/licenses/LICENSE-2.0

.. </legal notes>

parameters
==========

*)

METHOD testIsOverlapping
VAR_INPUT
	(* for the test it's the parameter ``address1`` *)
	address1		:PVOID;
	(* for the test it's the parameter ``address2`` *)
	address2		:PVOID;
	(* for the test it's the parameter ``sizeInBytes1`` *)
	sizeInBytes1	:UDINT;
	(* for the test it's the parameter ``sizeInBytes2`` *)
	sizeInBytes2	:UDINT;
END_VAR
VAR
	(* just the expectation if the assertion to test must be worng or true *)
	assertionIsWrong		:BOOL;
	(* contains the format string for the test message *)
	message					:Tc2_System.T_MaxString;
	(* TwinCAT printf with the test message *)
	messageStringBuilder	:Tc2_Utilities.FB_FormatString;
	(* contains adress of the stack of this method *)
	{attribute 'displaymode':='hex'}
	stackAddress			:__XWORD := ADR(stackAddress);
END_VAR
THIS^.assertorContainer.resetAssertor();

assertionIsWrong := address1 + sizeInBytes1 < address2 
					OR address2 + sizeInBytes2 < address1;

message := SEL(
	assertionIsWrong,
	'address1 is 16#%X, sizeInBytes is %d and address2 is 16#%X, sizeInBytes is %d, they are overlapping, assertion must be TRUE', 
	'address1 is 16#%X, sizeInBytes is %d and address2 is 16#%X, sizeInBytes is %d, they are not overlapping, assertion must be FALSE'
);
messageStringBuilder(
	sFormat := message,
	arg1 := THIS^.AnyToArg(address1),
	arg1 := THIS^.AnyToArg(sizeInBytes1),
	arg1 := THIS^.AnyToArg(address2),
	arg1 := THIS^.AnyToArg(sizeInBytes2),
);

THIS^.assertorContainer.assertor.assert.pointers.isOverlapping(
	address1 := address1,
	address2 := address2,
	sizeInBytes1 := sizeInBytes1,
	sizeInBytes2 := sizeInBytes2,
	message := ''
);

THIS^.AssertEquals_BOOL(
	Expected 	:= assertionIsWrong,
	Actual 		:= THIS^.assertorContainer.wasAssertionWrong,
	Message 	:= messageStringBuilder.sOut
);
END_METHOD

(*

short summary
==================
This test method tests ``assert.pointers.isValid``
method of CNM_AssertionInterfaces library, 
it provides the possibility to handover test data via parameter 

.. <legal notes>

legal notes
=================
| SPDX-FileCopyrightText: © 2022 ekvip automation GmbH <info@ekvip.de>
| SPDX-License-Identifier: Apache-2.0
| For details check: Apache-2.0_

.. _Apache-2.0: https://www.apache.org/licenses/LICENSE-2.0

.. </legal notes>

parameters
==========

*)

METHOD testIsValid
VAR_INPUT
	(* for the test it's the parameter ``address`` *)
	address		:PVOID;
	(* for the test it's the parameter ``sizeInBytes`` *)
	sizeInBytes	:UDINT;
	(* just the name of the pointer *)
	symbol		:Tc2_System.T_MaxString;
END_VAR
VAR
	(* just the expectation if the assertion to test must be worng or true *)
	assertionIsWrong		:BOOL;
	(* contains the format string for the test message *)
	message					:Tc2_System.T_MaxString;
	(* TwinCAT printf with the test message *)
	messageStringBuilder	:Tc2_Utilities.FB_FormatString;
	(* return value of Tc2_System.F_CheckMemoryArea *)
	memoryArea				:Tc2_System.E_TcMemoryArea;
	(*  return value of Tc2_System.F_CheckMemoryArea as string *)
	areaString				:Tc2_System.T_MaxString;
	(* contains adress of the stack of this method *)
	{attribute 'displaymode':='hex'}
	stackAddress	:__XWORD := ADR(stackAddress);
	{IF hasvalue (RegisterSize, '32')}
	(* lets try if it's possible to read something from the address *)
	validityTester			:POINTER TO BYTE;
	(* dummy variable with the value *)
	value					:BYTE;
	(* exception code *)
	e						:ExceptionCode;
	(* just to test it over all elemets *)
	count					:UDINT;
	{END_IF}
END_VAR
THIS^.assertorContainer.resetAssertor();

memoryArea	:= Tc2_System.F_CheckMemoryArea(address, sizeInBytes);
areaString	:= THIS^.memoryAreaToString(memoryArea);

{IF hasvalue (RegisterSize, '32')}
validityTester := address;
assertionIsWrong := ((
			(sizeInBytes <= THIS^.SIZE_ZERO
		) AND (
			address > THIS^.NULL_POINTER)
	) OR 
		//check for overflow
		address + sizeInBytes < address
);
__TRY
	IF (NOT assertionIsWrong) THEN
		FOR byteCount := 0 TO (sizeInBytes-1) DO
			value := validityTester[byteCount];
		END_FOR
	END_IF
__CATCH(e)
	assertionIsWrong := TRUE;
__ENDTRY
{ELSE}
assertionIsWrong := ((
		address = NULL_POINTER
	) OR (
		sizeInBytes <= NULL_POINTER
	) OR ((
		Tc2_System.F_CheckMemoryArea(pData := address, nSize := sizeInBytes) = Tc2_System.E_TcMemoryArea.Unknown
	) AND_THEN (
		address < (ABS(ADR(stackAddress) - MAX_STACK_SIZE)))
	) OR 
		//check for overflow
		address + sizeInBytes < address
);
{END_IF}

message := SEL(
	assertionIsWrong,
	'address is 16#%X ($'%s$') sizeInBytes is %d return value of Tc2_System.F_CheckMemoryArea is $'%s$' assertion must be TRUE', 
	'address is 16#%X ($'%s$') sizeInBytes is %d return value of Tc2_System.F_CheckMemoryArea is $'%s$' assertion must be FALSE'
);
messageStringBuilder(
	sFormat := message,
	arg1 := THIS^.AnyToArg(address),
	arg2 := THIS^.AnyToArg(symbol),
	arg3 := THIS^.AnyToArg(sizeInBytes),
	arg4 := THIS^.AnyToArg(areaString)
);

THIS^.assertorContainer.assertor.assert.pointers.isValid(
	address := address,
	sizeInBytes := sizeInBytes,
	message := ''
);

THIS^.AssertEquals_BOOL(
	Expected 	:= assertionIsWrong,
	Actual 		:= THIS^.assertorContainer.wasAssertionWrong,
	Message 	:= messageStringBuilder.sOut
);
END_METHOD

(*

short summary
==================
This test method tests ``assert.pointers.isWordAligned``
method of CNM_AssertionInterfaces library, 
it provides the possibility to handover test data via parameter
This test method uses a bit mask to verify correct memory alignment without duplicating the tested function.
(ex. for WORD: if bits 0 or 1 are set, the pointer is not aligned)

.. <legal notes>

legal notes
=================
| SPDX-FileCopyrightText: © 2022 ekvip automation GmbH <info@ekvip.de>
| SPDX-License-Identifier: Apache-2.0
| For details check: Apache-2.0_

.. _Apache-2.0: https://www.apache.org/licenses/LICENSE-2.0

.. </legal notes>

parameters
==========

*)

METHOD testIsWordAligned
VAR_INPUT
	(* for the test it's the parameter ``address`` *)
	address		:PVOID;
END_VAR
VAR
	(* just the expectation if the assertion to test must be worng or true *)
	assertionIsWrong		:BOOL;
	(* contains the format string for the test message *)
	message					:Tc2_System.T_MaxString;
	(* TwinCAT printf with the test message *)
	messageStringBuilder	:Tc2_Utilities.FB_FormatString;
	(* contains adress of the stack of this method *)
	{attribute 'displaymode':='hex'}
	stackAddress			:__XWORD := ADR(stackAddress);
END_VAR
VAR CONSTANT
	(* used to check if pointer is aligned *)
	{attribute 'displaymode':='hex'}
	alignmentMask 			:DWORD := 16#2;
END_VAR
THIS^.assertorContainer.resetAssertor();

assertionIsWrong := (alignmentMask AND address) <> 0;

message := SEL(
	assertionIsWrong,
	'address is 16#%X and should be aligned, assertion must be TRUE', 
	'address is 16#%X and should not be aligned, assertion must be FALSE'
);
messageStringBuilder(
	sFormat := message,
	arg1 := THIS^.AnyToArg(address),
);

THIS^.assertorContainer.assertor.assert.pointers.isWordAligned(
	address := address,
	message := ''
);

THIS^.AssertEquals_BOOL(
	Expected 	:= assertionIsWrong,
	Actual 		:= THIS^.assertorContainer.wasAssertionWrong,
	Message 	:= messageStringBuilder.sOut
);
END_METHOD

(*

short summary
==================
This test method tests ``assert.pointers.memoryAreaIsCnc``
method of CNM_AssertionInterfaces library, 
it provides the possibility to handover test data via parameter 

.. <legal notes>

legal notes
=================
| SPDX-FileCopyrightText: © 2022 ekvip automation GmbH <info@ekvip.de>
| SPDX-License-Identifier: Apache-2.0
| For details check: Apache-2.0_

.. _Apache-2.0: https://www.apache.org/licenses/LICENSE-2.0

.. </legal notes>

parameters
==========

*)

METHOD testMemoryAreaIsCnc
VAR_INPUT
	(* for the test it's the parameter ``address`` *)
	address		:PVOID;
	(* for the test it's the parameter ``sizeInBytes`` *)
	sizeInBytes	:UDINT;
	(* just the name of the pointer *)
	symbol		:Tc2_System.T_MaxString;
END_VAR
VAR
	(* just the expectation if the assertion to test must be worng or true *)
	assertionIsWrong		:BOOL;
	(* contains the format string for the test message *)
	message					:Tc2_System.T_MaxString;
	(* TwinCAT printf with the test message *)
	messageStringBuilder	:Tc2_Utilities.FB_FormatString;
	(* return value of Tc2_System.F_CheckMemoryArea *)
	memoryArea				:Tc2_System.E_TcMemoryArea;
	(*  return value of Tc2_System.F_CheckMemoryArea as string *)
	areaString				:Tc2_System.T_MaxString;
END_VAR
THIS^.assertorContainer.resetAssertor();

memoryArea	:= Tc2_System.F_CheckMemoryArea(address, sizeInBytes);
areaString	:= THIS^.memoryAreaToString(memoryArea);
assertionIsWrong := (memoryArea <> Tc2_System.E_TcMemoryArea.CNC);

message := SEL(
	assertionIsWrong,
	'address is 16#%X ($'%s$') sizeInBytes is %d return value of Tc2_System.F_CheckMemoryArea is $'%s$' assertion must be TRUE', 
	'address is 16#%X ($'%s$') sizeInBytes is %d return value of Tc2_System.F_CheckMemoryArea is $'%s$' assertion must be FALSE'
);
messageStringBuilder(
	sFormat := message,
	arg1 := THIS^.AnyToArg(address),
	arg2 := THIS^.AnyToArg(symbol),
	arg3 := THIS^.AnyToArg(sizeInBytes),
	arg4 := THIS^.AnyToArg(areaString)
);

THIS^.assertorContainer.assertor.assert.pointers.memoryAreaIsCnc(
	address := address,
	sizeInBytes := sizeInBytes,
	message := ''
);

THIS^.AssertEquals_BOOL(
	Expected 	:= assertionIsWrong,
	Actual 		:= THIS^.assertorContainer.wasAssertionWrong,
	Message 	:= messageStringBuilder.sOut
);
END_METHOD

(*

short summary
==================
This test method tests ``assert.pointers.memoryAreaIsDynamic``
method of CNM_AssertionInterfaces library, 
it provides the possibility to handover test data via parameter 

.. <legal notes>

legal notes
=================
| SPDX-FileCopyrightText: © 2022 ekvip automation GmbH <info@ekvip.de>
| SPDX-License-Identifier: Apache-2.0
| For details check: Apache-2.0_

.. _Apache-2.0: https://www.apache.org/licenses/LICENSE-2.0

.. </legal notes>

parameters
==========

*)

METHOD testMemoryAreaIsDynamic
VAR_INPUT
	(* for the test it's the parameter ``address`` *)
	address		:PVOID;
	(* for the test it's the parameter ``sizeInBytes`` *)
	sizeInBytes	:UDINT;
	(* just the name of the pointer *)
	symbol		:Tc2_System.T_MaxString;
END_VAR
VAR
	(* just the expectation if the assertion to test must be worng or true *)
	assertionIsWrong		:BOOL;
	(* contains the format string for the test message *)
	message					:Tc2_System.T_MaxString;
	(* TwinCAT printf with the test message *)
	messageStringBuilder	:Tc2_Utilities.FB_FormatString;
	(* return value of Tc2_System.F_CheckMemoryArea *)
	memoryArea				:Tc2_System.E_TcMemoryArea;
	(*  return value of Tc2_System.F_CheckMemoryArea as string *)
	areaString				:Tc2_System.T_MaxString;
END_VAR
THIS^.assertorContainer.resetAssertor();

memoryArea	:= Tc2_System.F_CheckMemoryArea(address, sizeInBytes);
areaString	:= THIS^.memoryAreaToString(memoryArea);
assertionIsWrong := (memoryArea <> Tc2_System.E_TcMemoryArea.Dynamic);

message := SEL(
	assertionIsWrong,
	'address is 16#%X ($'%s$') sizeInBytes is %d return value of Tc2_System.F_CheckMemoryArea is $'%s$' assertion must be TRUE', 
	'address is 16#%X ($'%s$') sizeInBytes is %d return value of Tc2_System.F_CheckMemoryArea is $'%s$' assertion must be FALSE'
);
messageStringBuilder(
	sFormat := message,
	arg1 := THIS^.AnyToArg(address),
	arg2 := THIS^.AnyToArg(symbol),
	arg3 := THIS^.AnyToArg(sizeInBytes),
	arg4 := THIS^.AnyToArg(areaString)
);

THIS^.assertorContainer.assertor.assert.pointers.memoryAreaIsDynamic(
	address := address,
	sizeInBytes := sizeInBytes,
	message := ''
);

THIS^.AssertEquals_BOOL(
	Expected 	:= assertionIsWrong,
	Actual 		:= THIS^.assertorContainer.wasAssertionWrong,
	Message 	:= messageStringBuilder.sOut
);
END_METHOD

(*

short summary
==================
This test method tests ``assert.pointers.memoryAreaIsNotCnc``
method of CNM_AssertionInterfaces library, 
it provides the possibility to handover test data via parameter 

.. <legal notes>

legal notes
=================
| SPDX-FileCopyrightText: © 2022 ekvip automation GmbH <info@ekvip.de>
| SPDX-License-Identifier: Apache-2.0
| For details check: Apache-2.0_

.. _Apache-2.0: https://www.apache.org/licenses/LICENSE-2.0

.. </legal notes>

parameters
==========

*)

METHOD testMemoryAreaIsNotCnc
VAR_INPUT
	(* for the test it's the parameter ``address`` *)
	address		:PVOID;
	(* for the test it's the parameter ``sizeInBytes`` *)
	sizeInBytes	:UDINT;
	(* just the name of the pointer *)
	symbol		:Tc2_System.T_MaxString;
END_VAR
VAR
	(* just the expectation if the assertion to test must be worng or true *)
	assertionIsWrong		:BOOL;
	(* contains the format string for the test message *)
	message					:Tc2_System.T_MaxString;
	(* TwinCAT printf with the test message *)
	messageStringBuilder	:Tc2_Utilities.FB_FormatString;
	(* return value of Tc2_System.F_CheckMemoryArea *)
	memoryArea				:Tc2_System.E_TcMemoryArea;
	(*  return value of Tc2_System.F_CheckMemoryArea as string *)
	areaString				:Tc2_System.T_MaxString;
END_VAR
THIS^.assertorContainer.resetAssertor();

memoryArea	:= Tc2_System.F_CheckMemoryArea(address, sizeInBytes);
areaString	:= THIS^.memoryAreaToString(memoryArea);
assertionIsWrong := (memoryArea = Tc2_System.E_TcMemoryArea.CNC);

message := SEL(
	assertionIsWrong,
	'address is 16#%X ($'%s$') sizeInBytes is %d return value of Tc2_System.F_CheckMemoryArea is $'%s$' assertion must be TRUE', 
	'address is 16#%X ($'%s$') sizeInBytes is %d return value of Tc2_System.F_CheckMemoryArea is $'%s$' assertion must be FALSE'
);
messageStringBuilder(
	sFormat := message,
	arg1 := THIS^.AnyToArg(address),
	arg2 := THIS^.AnyToArg(symbol),
	arg3 := THIS^.AnyToArg(sizeInBytes),
	arg4 := THIS^.AnyToArg(areaString)
);

THIS^.assertorContainer.assertor.assert.pointers.memoryAreaIsNotCnc(
	address := address,
	sizeInBytes := sizeInBytes,
	message := ''
);

THIS^.AssertEquals_BOOL(
	Expected 	:= assertionIsWrong,
	Actual 		:= THIS^.assertorContainer.wasAssertionWrong,
	Message 	:= messageStringBuilder.sOut
);
END_METHOD

(*

short summary
==================
This test method tests ``assert.pointers.memoryAreaIsNotDynamic``
method of CNM_AssertionInterfaces library, 
it provides the possibility to handover test data via parameter 

.. <legal notes>

legal notes
=================
| SPDX-FileCopyrightText: © 2022 ekvip automation GmbH <info@ekvip.de>
| SPDX-License-Identifier: Apache-2.0
| For details check: Apache-2.0_

.. _Apache-2.0: https://www.apache.org/licenses/LICENSE-2.0

.. </legal notes>

parameters
==========

*)

METHOD testMemoryAreaIsNotDynamic
VAR_INPUT
	(* for the test it's the parameter ``address`` *)
	address		:PVOID;
	(* for the test it's the parameter ``sizeInBytes`` *)
	sizeInBytes	:UDINT;
	(* just the name of the pointer *)
	symbol		:Tc2_System.T_MaxString;
END_VAR
VAR
	(* just the expectation if the assertion to test must be worng or true *)
	assertionIsWrong		:BOOL;
	(* contains the format string for the test message *)
	message					:Tc2_System.T_MaxString;
	(* TwinCAT printf with the test message *)
	messageStringBuilder	:Tc2_Utilities.FB_FormatString;
	(* return value of Tc2_System.F_CheckMemoryArea *)
	memoryArea				:Tc2_System.E_TcMemoryArea;
	(*  return value of Tc2_System.F_CheckMemoryArea as string *)
	areaString				:Tc2_System.T_MaxString;
END_VAR
THIS^.assertorContainer.resetAssertor();

memoryArea	:= Tc2_System.F_CheckMemoryArea(address, sizeInBytes);
areaString	:= THIS^.memoryAreaToString(memoryArea);
assertionIsWrong := (memoryArea = Tc2_System.E_TcMemoryArea.Dynamic);

message := SEL(
	assertionIsWrong,
	'address is 16#%X ($'%s$') sizeInBytes is %d return value of Tc2_System.F_CheckMemoryArea is $'%s$' assertion must be TRUE', 
	'address is 16#%X ($'%s$') sizeInBytes is %d return value of Tc2_System.F_CheckMemoryArea is $'%s$' assertion must be FALSE'
);
messageStringBuilder(
	sFormat := message,
	arg1 := THIS^.AnyToArg(address),
	arg2 := THIS^.AnyToArg(symbol),
	arg3 := THIS^.AnyToArg(sizeInBytes),
	arg4 := THIS^.AnyToArg(areaString)
);

THIS^.assertorContainer.assertor.assert.pointers.memoryAreaIsNotDynamic(
	address := address,
	sizeInBytes := sizeInBytes,
	message := ''
);

THIS^.AssertEquals_BOOL(
	Expected 	:= assertionIsWrong,
	Actual 		:= THIS^.assertorContainer.wasAssertionWrong,
	Message 	:= messageStringBuilder.sOut
);
END_METHOD

(*

short summary
==================
This test method tests ``assert.pointers.memoryAreaIsNotStatic``
method of CNM_AssertionInterfaces library, 
it provides the possibility to handover test data via parameter 

.. <legal notes>

legal notes
=================
| SPDX-FileCopyrightText: © 2022 ekvip automation GmbH <info@ekvip.de>
| SPDX-License-Identifier: Apache-2.0
| For details check: Apache-2.0_

.. _Apache-2.0: https://www.apache.org/licenses/LICENSE-2.0

.. </legal notes>

parameters
==========

*)

METHOD testMemoryAreaIsNotStatic
VAR_INPUT
	(* for the test it's the parameter ``address`` *)
	address		:PVOID;
	(* for the test it's the parameter ``sizeInBytes`` *)
	sizeInBytes	:UDINT;
	(* just the name of the pointer *)
	symbol		:Tc2_System.T_MaxString;
END_VAR
VAR
	(* just the expectation if the assertion to test must be worng or true *)
	assertionIsWrong		:BOOL;
	(* contains the format string for the test message *)
	message					:Tc2_System.T_MaxString;
	(* TwinCAT printf with the test message *)
	messageStringBuilder	:Tc2_Utilities.FB_FormatString;
	(* return value of Tc2_System.F_CheckMemoryArea *)
	memoryArea				:Tc2_System.E_TcMemoryArea;
	(*  return value of Tc2_System.F_CheckMemoryArea as string *)
	areaString				:Tc2_System.T_MaxString;
END_VAR
THIS^.assertorContainer.resetAssertor();

memoryArea	:= Tc2_System.F_CheckMemoryArea(address, sizeInBytes);
areaString	:= THIS^.memoryAreaToString(memoryArea);
assertionIsWrong := (memoryArea = Tc2_System.E_TcMemoryArea.Static);

message := SEL(
	assertionIsWrong,
	'address is 16#%X ($'%s$') sizeInBytes is %d return value of Tc2_System.F_CheckMemoryArea is $'%s$' assertion must be TRUE', 
	'address is 16#%X ($'%s$') sizeInBytes is %d return value of Tc2_System.F_CheckMemoryArea is $'%s$' assertion must be FALSE'
);
messageStringBuilder(
	sFormat := message,
	arg1 := THIS^.AnyToArg(address),
	arg2 := THIS^.AnyToArg(symbol),
	arg3 := THIS^.AnyToArg(sizeInBytes),
	arg4 := THIS^.AnyToArg(areaString)
);

THIS^.assertorContainer.assertor.assert.pointers.memoryAreaIsNotStatic(
	address := address,
	sizeInBytes := sizeInBytes,
	message := ''
);

THIS^.AssertEquals_BOOL(
	Expected 	:= assertionIsWrong,
	Actual 		:= THIS^.assertorContainer.wasAssertionWrong,
	Message 	:= messageStringBuilder.sOut
);
END_METHOD

(*

short summary
==================
This test method tests ``assert.pointers.memoryAreaIsNotUnkown``
method of CNM_AssertionInterfaces library, 
it provides the possibility to handover test data via parameter 

.. <legal notes>

legal notes
=================
| SPDX-FileCopyrightText: © 2022 ekvip automation GmbH <info@ekvip.de>
| SPDX-License-Identifier: Apache-2.0
| For details check: Apache-2.0_

.. _Apache-2.0: https://www.apache.org/licenses/LICENSE-2.0

.. </legal notes>

parameters
==========

*)

METHOD testMemoryAreaIsNotUnknown
VAR_INPUT
	(* for the test it's the parameter ``address`` *)
	address		:PVOID;
	(* for the test it's the parameter ``sizeInBytes`` *)
	sizeInBytes	:UDINT;
	(* just the name of the pointer *)
	symbol		:Tc2_System.T_MaxString;
END_VAR
VAR
	(* just the expectation if the assertion to test must be worng or true *)
	assertionIsWrong		:BOOL;
	(* contains the format string for the test message *)
	message					:Tc2_System.T_MaxString;
	(* TwinCAT printf with the test message *)
	messageStringBuilder	:Tc2_Utilities.FB_FormatString;
	(* return value of Tc2_System.F_CheckMemoryArea *)
	memoryArea				:Tc2_System.E_TcMemoryArea;
	(*  return value of Tc2_System.F_CheckMemoryArea as string *)
	areaString				:Tc2_System.T_MaxString;
END_VAR
THIS^.assertorContainer.resetAssertor();

memoryArea	:= Tc2_System.F_CheckMemoryArea(address, sizeInBytes);
areaString	:= THIS^.memoryAreaToString(memoryArea);
assertionIsWrong := (memoryArea = Tc2_System.E_TcMemoryArea.Unknown);

message := SEL(
	assertionIsWrong,
	'address is 16#%X ($'%s$') sizeInBytes is %d return value of Tc2_System.F_CheckMemoryArea is $'%s$' assertion must be TRUE', 
	'address is 16#%X ($'%s$') sizeInBytes is %d return value of Tc2_System.F_CheckMemoryArea is $'%s$' assertion must be FALSE'
);
messageStringBuilder(
	sFormat := message,
	arg1 := THIS^.AnyToArg(address),
	arg2 := THIS^.AnyToArg(symbol),
	arg3 := THIS^.AnyToArg(sizeInBytes),
	arg4 := THIS^.AnyToArg(areaString)
);

THIS^.assertorContainer.assertor.assert.pointers.memoryAreaIsNotUnkown(
	address := address,
	sizeInBytes := sizeInBytes,
	message := ''
);

THIS^.AssertEquals_BOOL(
	Expected 	:= assertionIsWrong,
	Actual 		:= THIS^.assertorContainer.wasAssertionWrong,
	Message 	:= messageStringBuilder.sOut
);
END_METHOD

(*

short summary
==================
This test method tests ``assert.pointers.memoryAreaIsStatic``
method of CNM_AssertionInterfaces library, 
it provides the possibility to handover test data via parameter 

.. <legal notes>

legal notes
=================
| SPDX-FileCopyrightText: © 2022 ekvip automation GmbH <info@ekvip.de>
| SPDX-License-Identifier: Apache-2.0
| For details check: Apache-2.0_

.. _Apache-2.0: https://www.apache.org/licenses/LICENSE-2.0

.. </legal notes>

parameters
==========

*)

METHOD testMemoryAreaIsStatic
VAR_INPUT
	(* for the test it's the parameter ``address`` *)
	address		:PVOID;
	(* for the test it's the parameter ``sizeInBytes`` *)
	sizeInBytes	:UDINT;
	(* just the name of the pointer *)
	symbol		:Tc2_System.T_MaxString;
END_VAR
VAR
	(* just the expectation if the assertion to test must be worng or true *)
	assertionIsWrong		:BOOL;
	(* contains the format string for the test message *)
	message					:Tc2_System.T_MaxString;
	(* TwinCAT printf with the test message *)
	messageStringBuilder	:Tc2_Utilities.FB_FormatString;
	(* return value of Tc2_System.F_CheckMemoryArea *)
	memoryArea				:Tc2_System.E_TcMemoryArea;
	(*  return value of Tc2_System.F_CheckMemoryArea as string *)
	areaString				:Tc2_System.T_MaxString;
END_VAR
THIS^.assertorContainer.resetAssertor();

memoryArea	:= Tc2_System.F_CheckMemoryArea(address, sizeInBytes);
areaString	:= THIS^.memoryAreaToString(memoryArea);
assertionIsWrong := (memoryArea <> Tc2_System.E_TcMemoryArea.Static);

message := SEL(
	assertionIsWrong,
	'address is 16#%X ($'%s$') sizeInBytes is %d return value of Tc2_System.F_CheckMemoryArea is $'%s$' assertion must be TRUE', 
	'address is 16#%X ($'%s$') sizeInBytes is %d return value of Tc2_System.F_CheckMemoryArea is $'%s$' assertion must be FALSE'
);
messageStringBuilder(
	sFormat := message,
	arg1 := THIS^.AnyToArg(address),
	arg2 := THIS^.AnyToArg(symbol),
	arg3 := THIS^.AnyToArg(sizeInBytes),
	arg4 := THIS^.AnyToArg(areaString)
);

THIS^.assertorContainer.assertor.assert.pointers.memoryAreaIsStatic(
	address := address,
	sizeInBytes := sizeInBytes,
	message := ''
);

THIS^.AssertEquals_BOOL(
	Expected 	:= assertionIsWrong,
	Actual 		:= THIS^.assertorContainer.wasAssertionWrong,
	Message 	:= messageStringBuilder.sOut
);
END_METHOD

(*

short summary
==================
This test method tests ``assert.pointers.memoryAreaIsUnkown``
method of CNM_AssertionInterfaces library, 
it provides the possibility to handover test data via parameter 

.. <legal notes>

legal notes
=================
| SPDX-FileCopyrightText: © 2022 ekvip automation GmbH <info@ekvip.de>
| SPDX-License-Identifier: Apache-2.0
| For details check: Apache-2.0_

.. _Apache-2.0: https://www.apache.org/licenses/LICENSE-2.0

.. </legal notes>

parameters
==========

*)

METHOD testMemoryAreaIsUnknown
VAR_INPUT
	(* for the test it's the parameter ``address`` *)
	address		:PVOID;
	(* for the test it's the parameter ``sizeInBytes`` *)
	sizeInBytes	:UDINT;
	(* just the name of the pointer *)
	symbol		:Tc2_System.T_MaxString;
END_VAR
VAR
	(* just the expectation if the assertion to test must be worng or true *)
	assertionIsWrong		:BOOL;
	(* contains the format string for the test message *)
	message					:Tc2_System.T_MaxString;
	(* TwinCAT printf with the test message *)
	messageStringBuilder	:Tc2_Utilities.FB_FormatString;
	(* return value of Tc2_System.F_CheckMemoryArea *)
	memoryArea				:Tc2_System.E_TcMemoryArea;
	(*  return value of Tc2_System.F_CheckMemoryArea as string *)
	areaString				:Tc2_System.T_MaxString;
END_VAR
THIS^.assertorContainer.resetAssertor();

memoryArea	:= Tc2_System.F_CheckMemoryArea(address, sizeInBytes);
areaString	:= THIS^.memoryAreaToString(memoryArea);
assertionIsWrong := (memoryArea <> Tc2_System.E_TcMemoryArea.Unknown);

message := SEL(
	assertionIsWrong,
	'address is 16#%X ($'%s$') sizeInBytes is %d return value of Tc2_System.F_CheckMemoryArea is $'%s$' assertion must be TRUE', 
	'address is 16#%X ($'%s$') sizeInBytes is %d return value of Tc2_System.F_CheckMemoryArea is $'%s$' assertion must be FALSE'
);
messageStringBuilder(
	sFormat := message,
	arg1 := THIS^.AnyToArg(address),
	arg2 := THIS^.AnyToArg(symbol),
	arg3 := THIS^.AnyToArg(sizeInBytes),
	arg4 := THIS^.AnyToArg(areaString)
);

THIS^.assertorContainer.assertor.assert.pointers.memoryAreaIsUnkown(
	address := address,
	sizeInBytes := sizeInBytes,
	message := ''
);

THIS^.AssertEquals_BOOL(
	Expected 	:= assertionIsWrong,
	Actual 		:= THIS^.assertorContainer.wasAssertionWrong,
	Message 	:= messageStringBuilder.sOut
);
END_METHOD

(*

short summary
==================
This test method tests ``assert.pointers.isNotEqualTo``
method of CNM_AssertionInterfaces library, 
it provides the possibility to handover test data via parameter 


.. <legal notes>

legal notes
=================
| SPDX-FileCopyrightText: © 2022 ekvip automation GmbH <info@ekvip.de>
| SPDX-License-Identifier: Apache-2.0
| For details check: Apache-2.0_

.. _Apache-2.0: https://www.apache.org/licenses/LICENSE-2.0

.. </legal notes>

parameters
==========

*)

METHOD testNotIsEqualTo
VAR_INPUT
	(* for the test it's the parameter ``address1`` *)
	address1	:PVOID;
	(* for the test it's the parameter ``address2`` *)
	address2	:PVOID;
END_VAR
VAR
	(* just the expectation if the assertion to test must be worng or true *)
	assertionIsWrong		:BOOL;
	(* contains the format string for the test message *)
	message					:Tc2_System.T_MaxString;
	(* TwinCAT printf with the test message *)
	messageStringBuilder	:Tc2_Utilities.FB_FormatString;
END_VAR
THIS^.assertorContainer.resetAssertor();

assertionIsWrong := (address1 = address2);
message := SEL(
	assertionIsWrong,
	'address1 is 16#%X address2 is 16#%X assertion must be TRUE', 
	'address1 is 16#%X address2 is 16#%X assertion must be FALSE'
);
messageStringBuilder(
	sFormat := message,
	arg1 := THIS^.AnyToArg(address1),
	arg2 := THIS^.AnyToArg(address2)
);

THIS^.assertorContainer.assertor.assert.pointers.isNotEqualTo(
	address1 := address1,
	address2 := address2,
	message := ''
);

THIS^.AssertEquals_BOOL(
	Expected 	:= assertionIsWrong,
	Actual 		:= THIS^.assertorContainer.wasAssertionWrong,
	Message 	:= messageStringBuilder.sOut
);
END_METHOD

END_FUNCTION_BLOCK

// ---- AssertionTester/AssertionTests/StringAssertions/classes/UnicodeUtf16StringAssertionTests.TcPOU

(*
short summary
==================
This class tests all methods of Unicode string assertions
with various UTF-16 string combinations as input and checks expected 
outputs are satisfied or not

.. <legal notes>

legal notes
=================
| SPDX-FileCopyrightText: © 2022 ekvip automation GmbH <info@ekvip.de>
| SPDX-License-Identifier: Apache-2.0
| For details check: Apache-2.0_

.. _Apache-2.0: https://www.apache.org/licenses/LICENSE-2.0

.. </legal notes>

methods and properties
======================

*)


FUNCTION_BLOCK UnicodeUtf16StringAssertionTests EXTENDS AbstractAssertorTest
VAR

END_VAR
VAR CONSTANT
	(* prefix to unify the test names *)
	TEST_NAME_PREFIX :STRING := 'assert.string.unicode(utf16).';
END_VAR

THIS^.runIsEmpty();
THIS^.runIsNotEmpty();
THIS^.runContains();
THIS^.runContainsNo();
THIS^.runEndsWith();
THIS^.runStartsWith();
THIS^.runIsEqualTo();
THIS^.runIsNotEqualTo();
THIS^.runLengthIsBetween();
THIS^.runLengthIsExact();
THIS^.runLengthIsMax();
THIS^.runLengthIsMin();

(*

short summary
==================
This test method is a helper function to create a unified test name

.. <legal notes>

legal notes
=================
| SPDX-FileCopyrightText: © 2022 ekvip automation GmbH <info@ekvip.de>
| SPDX-License-Identifier: Apache-2.0
| For details check: Apache-2.0_

.. _Apache-2.0: https://www.apache.org/licenses/LICENSE-2.0

.. </legal notes>

parameters
==========

*)

METHOD PROTECTED getTestNameFor :Tc2_System.T_MaxString
VAR_INPUT
	(* name of the method to test, to create a unified test name *)
	nameOfMethodToTest	:Tc2_System.T_MaxString;
END_VAR
getTestNameFor := Tc2_Standard.CONCAT(THIS^.TEST_NAME_PREFIX, nameOfMethodToTest);
END_METHOD

(*
short summary
==================
This test method tests ``assert.string.unicode.contains``
method of CNM_AssertionInterfaces library with various inputs

.. <legal notes>

legal notes
=================
| SPDX-FileCopyrightText: © 2022 ekvip automation GmbH <info@ekvip.de>
| SPDX-License-Identifier: Apache-2.0
| For details check: Apache-2.0_

.. _Apache-2.0: https://www.apache.org/licenses/LICENSE-2.0

.. </legal notes>

*)


METHOD runContains : BOOL
VAR_INPUT
END_VAR
RETURN (NOT TcUnit.TEST_ORDERED(THIS^.getTestNameFor('contains')));

